   STATUS[640].EXT.AlarmPrsent := FALSE;
   STATUS[640].EXT.AlarmFailUnAck := FALSE;
   STATUS[640].Status := 0;
   STATUS[640].TimeStamp := 16#0000;
   STATUS[641].VALUE := 0.0;
   STATUS[641].TRIGVALUE := 0.0;
   STATUS[641].EXT.AlarmWarnUnAck := FALSE;
   STATUS[641].EXT.AckRequired := FALSE;
   STATUS[641].EXT.Maintanence := FALSE;
   STATUS[641].EXT.Operation := FALSE;
   STATUS[641].EXT.Forced := FALSE;
   STATUS[641].EXT.BIT29 := FALSE;
   STATUS[641].EXT.BIT30 := FALSE;
   STATUS[641].EXT.BIT31 := FALSE;
   STATUS[641].EXT.ModeBit1 := FALSE;
   STATUS[641].EXT.ModeBit2 := FALSE;
   STATUS[641].EXT.ModeBit3 := FALSE;
   STATUS[641].EXT.BIT19 := FALSE;
   STATUS[641].EXT.BIT20 := FALSE;
   STATUS[641].EXT.AlarmSuppressed := FALSE;
   STATUS[641].EXT.AlarmPrsent := FALSE;
   STATUS[641].EXT.AlarmFailUnAck := FALSE;
   STATUS[641].Status := 0;
   STATUS[641].TimeStamp := 16#0000;
   STATUS[642].VALUE := 0.0;
   STATUS[642].TRIGVALUE := 0.0;
   STATUS[642].EXT.AlarmWarnUnAck := FALSE;
   STATUS[642].EXT.AckRequired := FALSE;
   STATUS[642].EXT.Maintanence := FALSE;
   STATUS[642].EXT.Operation := FALSE;
   STATUS[642].EXT.Forced := FALSE;
   STATUS[642].EXT.BIT29 := FALSE;
   STATUS[642].EXT.BIT30 := FALSE;
   STATUS[642].EXT.BIT31 := FALSE;
   STATUS[642].EXT.ModeBit1 := FALSE;
   STATUS[642].EXT.ModeBit2 := FALSE;
   STATUS[642].EXT.ModeBit3 := FALSE;
   STATUS[642].EXT.BIT19 := FALSE;
   STATUS[642].EXT.BIT20 := FALSE;
   STATUS[642].EXT.AlarmSuppressed := FALSE;
   STATUS[642].EXT.AlarmPrsent := FALSE;
   STATUS[642].EXT.AlarmFailUnAck := FALSE;
   STATUS[642].Status := 0;
   STATUS[642].TimeStamp := 16#0000;
   STATUS[643].VALUE := 0.0;
   STATUS[643].TRIGVALUE := 0.0;
   STATUS[643].EXT.AlarmWarnUnAck := FALSE;
   STATUS[643].EXT.AckRequired := FALSE;
   STATUS[643].EXT.Maintanence := FALSE;
   STATUS[643].EXT.Operation := FALSE;
   STATUS[643].EXT.Forced := FALSE;
   STATUS[643].EXT.BIT29 := FALSE;
   STATUS[643].EXT.BIT30 := FALSE;
   STATUS[643].EXT.BIT31 := FALSE;
   STATUS[643].EXT.ModeBit1 := FALSE;
   STATUS[643].EXT.ModeBit2 := FALSE;
   STATUS[643].EXT.ModeBit3 := FALSE;
   STATUS[643].EXT.BIT19 := FALSE;
   STATUS[643].EXT.BIT20 := FALSE;
   STATUS[643].EXT.AlarmSuppressed := FALSE;
   STATUS[643].EXT.AlarmPrsent := FALSE;
   STATUS[643].EXT.AlarmFailUnAck := FALSE;
   STATUS[643].Status := 0;
   STATUS[643].TimeStamp := 16#0000;
   STATUS[644].VALUE := 0.0;
   STATUS[644].TRIGVALUE := 0.0;
   STATUS[644].EXT.AlarmWarnUnAck := FALSE;
   STATUS[644].EXT.AckRequired := FALSE;
   STATUS[644].EXT.Maintanence := FALSE;
   STATUS[644].EXT.Operation := FALSE;
   STATUS[644].EXT.Forced := FALSE;
   STATUS[644].EXT.BIT29 := FALSE;
   STATUS[644].EXT.BIT30 := FALSE;
   STATUS[644].EXT.BIT31 := FALSE;
   STATUS[644].EXT.ModeBit1 := FALSE;
   STATUS[644].EXT.ModeBit2 := FALSE;
   STATUS[644].EXT.ModeBit3 := FALSE;
   STATUS[644].EXT.BIT19 := FALSE;
   STATUS[644].EXT.BIT20 := FALSE;
   STATUS[644].EXT.AlarmSuppressed := FALSE;
   STATUS[644].EXT.AlarmPrsent := FALSE;
   STATUS[644].EXT.AlarmFailUnAck := FALSE;
   STATUS[644].Status := 0;
   STATUS[644].TimeStamp := 16#0000;
   STATUS[645].VALUE := 0.0;
   STATUS[645].TRIGVALUE := 0.0;
   STATUS[645].EXT.AlarmWarnUnAck := FALSE;
   STATUS[645].EXT.AckRequired := FALSE;
   STATUS[645].EXT.Maintanence := FALSE;
   STATUS[645].EXT.Operation := FALSE;
   STATUS[645].EXT.Forced := FALSE;
   STATUS[645].EXT.BIT29 := FALSE;
   STATUS[645].EXT.BIT30 := FALSE;
   STATUS[645].EXT.BIT31 := FALSE;
   STATUS[645].EXT.ModeBit1 := FALSE;
   STATUS[645].EXT.ModeBit2 := FALSE;
   STATUS[645].EXT.ModeBit3 := FALSE;
   STATUS[645].EXT.BIT19 := FALSE;
   STATUS[645].EXT.BIT20 := FALSE;
   STATUS[645].EXT.AlarmSuppressed := FALSE;
   STATUS[645].EXT.AlarmPrsent := FALSE;
   STATUS[645].EXT.AlarmFailUnAck := FALSE;
   STATUS[645].Status := 0;
   STATUS[645].TimeStamp := 16#0000;
   STATUS[646].VALUE := 0.0;
   STATUS[646].TRIGVALUE := 0.0;
   STATUS[646].EXT.AlarmWarnUnAck := FALSE;
   STATUS[646].EXT.AckRequired := FALSE;
   STATUS[646].EXT.Maintanence := FALSE;
   STATUS[646].EXT.Operation := FALSE;
   STATUS[646].EXT.Forced := FALSE;
   STATUS[646].EXT.BIT29 := FALSE;
   STATUS[646].EXT.BIT30 := FALSE;
   STATUS[646].EXT.BIT31 := FALSE;
   STATUS[646].EXT.ModeBit1 := FALSE;
   STATUS[646].EXT.ModeBit2 := FALSE;
   STATUS[646].EXT.ModeBit3 := FALSE;
   STATUS[646].EXT.BIT19 := FALSE;
   STATUS[646].EXT.BIT20 := FALSE;
   STATUS[646].EXT.AlarmSuppressed := FALSE;
   STATUS[646].EXT.AlarmPrsent := FALSE;
   STATUS[646].EXT.AlarmFailUnAck := FALSE;
   STATUS[646].Status := 0;
   STATUS[646].TimeStamp := 16#0000;
   STATUS[647].VALUE := 0.0;
   STATUS[647].TRIGVALUE := 0.0;
   STATUS[647].EXT.AlarmWarnUnAck := FALSE;
   STATUS[647].EXT.AckRequired := FALSE;
   STATUS[647].EXT.Maintanence := FALSE;
   STATUS[647].EXT.Operation := FALSE;
   STATUS[647].EXT.Forced := FALSE;
   STATUS[647].EXT.BIT29 := FALSE;
   STATUS[647].EXT.BIT30 := FALSE;
   STATUS[647].EXT.BIT31 := FALSE;
   STATUS[647].EXT.ModeBit1 := FALSE;
   STATUS[647].EXT.ModeBit2 := FALSE;
   STATUS[647].EXT.ModeBit3 := FALSE;
   STATUS[647].EXT.BIT19 := FALSE;
   STATUS[647].EXT.BIT20 := FALSE;
   STATUS[647].EXT.AlarmSuppressed := FALSE;
   STATUS[647].EXT.AlarmPrsent := FALSE;
   STATUS[647].EXT.AlarmFailUnAck := FALSE;
   STATUS[647].Status := 0;
   STATUS[647].TimeStamp := 16#0000;
   STATUS[648].VALUE := 0.0;
   STATUS[648].TRIGVALUE := 0.0;
   STATUS[648].EXT.AlarmWarnUnAck := FALSE;
   STATUS[648].EXT.AckRequired := FALSE;
   STATUS[648].EXT.Maintanence := FALSE;
   STATUS[648].EXT.Operation := FALSE;
   STATUS[648].EXT.Forced := FALSE;
   STATUS[648].EXT.BIT29 := FALSE;
   STATUS[648].EXT.BIT30 := FALSE;
   STATUS[648].EXT.BIT31 := FALSE;
   STATUS[648].EXT.ModeBit1 := FALSE;
   STATUS[648].EXT.ModeBit2 := FALSE;
   STATUS[648].EXT.ModeBit3 := FALSE;
   STATUS[648].EXT.BIT19 := FALSE;
   STATUS[648].EXT.BIT20 := FALSE;
   STATUS[648].EXT.AlarmSuppressed := FALSE;
   STATUS[648].EXT.AlarmPrsent := FALSE;
   STATUS[648].EXT.AlarmFailUnAck := FALSE;
   STATUS[648].Status := 0;
   STATUS[648].TimeStamp := 16#0000;
   STATUS[649].VALUE := 0.0;
   STATUS[649].TRIGVALUE := 0.0;
   STATUS[649].EXT.AlarmWarnUnAck := FALSE;
   STATUS[649].EXT.AckRequired := FALSE;
   STATUS[649].EXT.Maintanence := FALSE;
   STATUS[649].EXT.Operation := FALSE;
   STATUS[649].EXT.Forced := FALSE;
   STATUS[649].EXT.BIT29 := FALSE;
   STATUS[649].EXT.BIT30 := FALSE;
   STATUS[649].EXT.BIT31 := FALSE;
   STATUS[649].EXT.ModeBit1 := FALSE;
   STATUS[649].EXT.ModeBit2 := FALSE;
   STATUS[649].EXT.ModeBit3 := FALSE;
   STATUS[649].EXT.BIT19 := FALSE;
   STATUS[649].EXT.BIT20 := FALSE;
   STATUS[649].EXT.AlarmSuppressed := FALSE;
   STATUS[649].EXT.AlarmPrsent := FALSE;
   STATUS[649].EXT.AlarmFailUnAck := FALSE;
   STATUS[649].Status := 0;
   STATUS[649].TimeStamp := 16#0000;
   STATUS[650].VALUE := 0.0;
   STATUS[650].TRIGVALUE := 0.0;
   STATUS[650].EXT.AlarmWarnUnAck := FALSE;
   STATUS[650].EXT.AckRequired := FALSE;
   STATUS[650].EXT.Maintanence := FALSE;
   STATUS[650].EXT.Operation := FALSE;
   STATUS[650].EXT.Forced := FALSE;
   STATUS[650].EXT.BIT29 := FALSE;
   STATUS[650].EXT.BIT30 := FALSE;
   STATUS[650].EXT.BIT31 := FALSE;
   STATUS[650].EXT.ModeBit1 := FALSE;
   STATUS[650].EXT.ModeBit2 := FALSE;
   STATUS[650].EXT.ModeBit3 := FALSE;
   STATUS[650].EXT.BIT19 := FALSE;
   STATUS[650].EXT.BIT20 := FALSE;
   STATUS[650].EXT.AlarmSuppressed := FALSE;
   STATUS[650].EXT.AlarmPrsent := FALSE;
   STATUS[650].EXT.AlarmFailUnAck := FALSE;
   STATUS[650].Status := 0;
   STATUS[650].TimeStamp := 16#0000;
   STATUS[651].VALUE := 0.0;
   STATUS[651].TRIGVALUE := 0.0;
   STATUS[651].EXT.AlarmWarnUnAck := FALSE;
   STATUS[651].EXT.AckRequired := FALSE;
   STATUS[651].EXT.Maintanence := FALSE;
   STATUS[651].EXT.Operation := FALSE;
   STATUS[651].EXT.Forced := FALSE;
   STATUS[651].EXT.BIT29 := FALSE;
   STATUS[651].EXT.BIT30 := FALSE;
   STATUS[651].EXT.BIT31 := FALSE;
   STATUS[651].EXT.ModeBit1 := FALSE;
   STATUS[651].EXT.ModeBit2 := FALSE;
   STATUS[651].EXT.ModeBit3 := FALSE;
   STATUS[651].EXT.BIT19 := FALSE;
   STATUS[651].EXT.BIT20 := FALSE;
   STATUS[651].EXT.AlarmSuppressed := FALSE;
   STATUS[651].EXT.AlarmPrsent := FALSE;
   STATUS[651].EXT.AlarmFailUnAck := FALSE;
   STATUS[651].Status := 0;
   STATUS[651].TimeStamp := 16#0000;
   STATUS[652].VALUE := 0.0;
   STATUS[652].TRIGVALUE := 0.0;
   STATUS[652].EXT.AlarmWarnUnAck := FALSE;
   STATUS[652].EXT.AckRequired := FALSE;
   STATUS[652].EXT.Maintanence := FALSE;
   STATUS[652].EXT.Operation := FALSE;
   STATUS[652].EXT.Forced := FALSE;
   STATUS[652].EXT.BIT29 := FALSE;
   STATUS[652].EXT.BIT30 := FALSE;
   STATUS[652].EXT.BIT31 := FALSE;
   STATUS[652].EXT.ModeBit1 := FALSE;
   STATUS[652].EXT.ModeBit2 := FALSE;
   STATUS[652].EXT.ModeBit3 := FALSE;
   STATUS[652].EXT.BIT19 := FALSE;
   STATUS[652].EXT.BIT20 := FALSE;
   STATUS[652].EXT.AlarmSuppressed := FALSE;
   STATUS[652].EXT.AlarmPrsent := FALSE;
   STATUS[652].EXT.AlarmFailUnAck := FALSE;
   STATUS[652].Status := 0;
   STATUS[652].TimeStamp := 16#0000;
   STATUS[653].VALUE := 0.0;
   STATUS[653].TRIGVALUE := 0.0;
   STATUS[653].EXT.AlarmWarnUnAck := FALSE;
   STATUS[653].EXT.AckRequired := FALSE;
   STATUS[653].EXT.Maintanence := FALSE;
   STATUS[653].EXT.Operation := FALSE;
   STATUS[653].EXT.Forced := FALSE;
   STATUS[653].EXT.BIT29 := FALSE;
   STATUS[653].EXT.BIT30 := FALSE;
   STATUS[653].EXT.BIT31 := FALSE;
   STATUS[653].EXT.ModeBit1 := FALSE;
   STATUS[653].EXT.ModeBit2 := FALSE;
   STATUS[653].EXT.ModeBit3 := FALSE;
   STATUS[653].EXT.BIT19 := FALSE;
   STATUS[653].EXT.BIT20 := FALSE;
   STATUS[653].EXT.AlarmSuppressed := FALSE;
   STATUS[653].EXT.AlarmPrsent := FALSE;
   STATUS[653].EXT.AlarmFailUnAck := FALSE;
   STATUS[653].Status := 0;
   STATUS[653].TimeStamp := 16#0000;
   STATUS[654].VALUE := 0.0;
   STATUS[654].TRIGVALUE := 0.0;
   STATUS[654].EXT.AlarmWarnUnAck := FALSE;
   STATUS[654].EXT.AckRequired := FALSE;
   STATUS[654].EXT.Maintanence := FALSE;
   STATUS[654].EXT.Operation := FALSE;
   STATUS[654].EXT.Forced := FALSE;
   STATUS[654].EXT.BIT29 := FALSE;
   STATUS[654].EXT.BIT30 := FALSE;
   STATUS[654].EXT.BIT31 := FALSE;
   STATUS[654].EXT.ModeBit1 := FALSE;
   STATUS[654].EXT.ModeBit2 := FALSE;
   STATUS[654].EXT.ModeBit3 := FALSE;
   STATUS[654].EXT.BIT19 := FALSE;
   STATUS[654].EXT.BIT20 := FALSE;
   STATUS[654].EXT.AlarmSuppressed := FALSE;
   STATUS[654].EXT.AlarmPrsent := FALSE;
   STATUS[654].EXT.AlarmFailUnAck := FALSE;
   STATUS[654].Status := 0;
   STATUS[654].TimeStamp := 16#0000;
   STATUS[655].VALUE := 0.0;
   STATUS[655].TRIGVALUE := 0.0;
   STATUS[655].EXT.AlarmWarnUnAck := FALSE;
   STATUS[655].EXT.AckRequired := FALSE;
   STATUS[655].EXT.Maintanence := FALSE;
   STATUS[655].EXT.Operation := FALSE;
   STATUS[655].EXT.Forced := FALSE;
   STATUS[655].EXT.BIT29 := FALSE;
   STATUS[655].EXT.BIT30 := FALSE;
   STATUS[655].EXT.BIT31 := FALSE;
   STATUS[655].EXT.ModeBit1 := FALSE;
   STATUS[655].EXT.ModeBit2 := FALSE;
   STATUS[655].EXT.ModeBit3 := FALSE;
   STATUS[655].EXT.BIT19 := FALSE;
   STATUS[655].EXT.BIT20 := FALSE;
   STATUS[655].EXT.AlarmSuppressed := FALSE;
   STATUS[655].EXT.AlarmPrsent := FALSE;
   STATUS[655].EXT.AlarmFailUnAck := FALSE;
   STATUS[655].Status := 0;
   STATUS[655].TimeStamp := 16#0000;
   STATUS[656].VALUE := 0.0;
   STATUS[656].TRIGVALUE := 0.0;
   STATUS[656].EXT.AlarmWarnUnAck := FALSE;
   STATUS[656].EXT.AckRequired := FALSE;
   STATUS[656].EXT.Maintanence := FALSE;
   STATUS[656].EXT.Operation := FALSE;
   STATUS[656].EXT.Forced := FALSE;
   STATUS[656].EXT.BIT29 := FALSE;
   STATUS[656].EXT.BIT30 := FALSE;
   STATUS[656].EXT.BIT31 := FALSE;
   STATUS[656].EXT.ModeBit1 := FALSE;
   STATUS[656].EXT.ModeBit2 := FALSE;
   STATUS[656].EXT.ModeBit3 := FALSE;
   STATUS[656].EXT.BIT19 := FALSE;
   STATUS[656].EXT.BIT20 := FALSE;
   STATUS[656].EXT.AlarmSuppressed := FALSE;
   STATUS[656].EXT.AlarmPrsent := FALSE;
   STATUS[656].EXT.AlarmFailUnAck := FALSE;
   STATUS[656].Status := 0;
   STATUS[656].TimeStamp := 16#0000;
   STATUS[657].VALUE := 0.0;
   STATUS[657].TRIGVALUE := 0.0;
   STATUS[657].EXT.AlarmWarnUnAck := FALSE;
   STATUS[657].EXT.AckRequired := FALSE;
   STATUS[657].EXT.Maintanence := FALSE;
   STATUS[657].EXT.Operation := FALSE;
   STATUS[657].EXT.Forced := FALSE;
   STATUS[657].EXT.BIT29 := FALSE;
   STATUS[657].EXT.BIT30 := FALSE;
   STATUS[657].EXT.BIT31 := FALSE;
   STATUS[657].EXT.ModeBit1 := FALSE;
   STATUS[657].EXT.ModeBit2 := FALSE;
   STATUS[657].EXT.ModeBit3 := FALSE;
   STATUS[657].EXT.BIT19 := FALSE;
   STATUS[657].EXT.BIT20 := FALSE;
   STATUS[657].EXT.AlarmSuppressed := FALSE;
   STATUS[657].EXT.AlarmPrsent := FALSE;
   STATUS[657].EXT.AlarmFailUnAck := FALSE;
   STATUS[657].Status := 0;
   STATUS[657].TimeStamp := 16#0000;
   STATUS[658].VALUE := 0.0;
   STATUS[658].TRIGVALUE := 0.0;
   STATUS[658].EXT.AlarmWarnUnAck := FALSE;
   STATUS[658].EXT.AckRequired := FALSE;
   STATUS[658].EXT.Maintanence := FALSE;
   STATUS[658].EXT.Operation := FALSE;
   STATUS[658].EXT.Forced := FALSE;
   STATUS[658].EXT.BIT29 := FALSE;
   STATUS[658].EXT.BIT30 := FALSE;
   STATUS[658].EXT.BIT31 := FALSE;
   STATUS[658].EXT.ModeBit1 := FALSE;
   STATUS[658].EXT.ModeBit2 := FALSE;
   STATUS[658].EXT.ModeBit3 := FALSE;
   STATUS[658].EXT.BIT19 := FALSE;
   STATUS[658].EXT.BIT20 := FALSE;
   STATUS[658].EXT.AlarmSuppressed := FALSE;
   STATUS[658].EXT.AlarmPrsent := FALSE;
   STATUS[658].EXT.AlarmFailUnAck := FALSE;
   STATUS[658].Status := 0;
   STATUS[658].TimeStamp := 16#0000;
   STATUS[659].VALUE := 0.0;
   STATUS[659].TRIGVALUE := 0.0;
   STATUS[659].EXT.AlarmWarnUnAck := FALSE;
   STATUS[659].EXT.AckRequired := FALSE;
   STATUS[659].EXT.Maintanence := FALSE;
   STATUS[659].EXT.Operation := FALSE;
   STATUS[659].EXT.Forced := FALSE;
   STATUS[659].EXT.BIT29 := FALSE;
   STATUS[659].EXT.BIT30 := FALSE;
   STATUS[659].EXT.BIT31 := FALSE;
   STATUS[659].EXT.ModeBit1 := FALSE;
   STATUS[659].EXT.ModeBit2 := FALSE;
   STATUS[659].EXT.ModeBit3 := FALSE;
   STATUS[659].EXT.BIT19 := FALSE;
   STATUS[659].EXT.BIT20 := FALSE;
   STATUS[659].EXT.AlarmSuppressed := FALSE;
   STATUS[659].EXT.AlarmPrsent := FALSE;
   STATUS[659].EXT.AlarmFailUnAck := FALSE;
   STATUS[659].Status := 0;
   STATUS[659].TimeStamp := 16#0000;
   STATUS[660].VALUE := 0.0;
   STATUS[660].TRIGVALUE := 0.0;
   STATUS[660].EXT.AlarmWarnUnAck := FALSE;
   STATUS[660].EXT.AckRequired := FALSE;
   STATUS[660].EXT.Maintanence := FALSE;
   STATUS[660].EXT.Operation := FALSE;
   STATUS[660].EXT.Forced := FALSE;
   STATUS[660].EXT.BIT29 := FALSE;
   STATUS[660].EXT.BIT30 := FALSE;
   STATUS[660].EXT.BIT31 := FALSE;
   STATUS[660].EXT.ModeBit1 := FALSE;
   STATUS[660].EXT.ModeBit2 := FALSE;
   STATUS[660].EXT.ModeBit3 := FALSE;
   STATUS[660].EXT.BIT19 := FALSE;
   STATUS[660].EXT.BIT20 := FALSE;
   STATUS[660].EXT.AlarmSuppressed := FALSE;
   STATUS[660].EXT.AlarmPrsent := FALSE;
   STATUS[660].EXT.AlarmFailUnAck := FALSE;
   STATUS[660].Status := 0;
   STATUS[660].TimeStamp := 16#0000;
   STATUS[661].VALUE := 0.0;
   STATUS[661].TRIGVALUE := 0.0;
   STATUS[661].EXT.AlarmWarnUnAck := FALSE;
   STATUS[661].EXT.AckRequired := FALSE;
   STATUS[661].EXT.Maintanence := FALSE;
   STATUS[661].EXT.Operation := FALSE;
   STATUS[661].EXT.Forced := FALSE;
   STATUS[661].EXT.BIT29 := FALSE;
   STATUS[661].EXT.BIT30 := FALSE;
   STATUS[661].EXT.BIT31 := FALSE;
   STATUS[661].EXT.ModeBit1 := FALSE;
   STATUS[661].EXT.ModeBit2 := FALSE;
   STATUS[661].EXT.ModeBit3 := FALSE;
   STATUS[661].EXT.BIT19 := FALSE;
   STATUS[661].EXT.BIT20 := FALSE;
   STATUS[661].EXT.AlarmSuppressed := FALSE;
   STATUS[661].EXT.AlarmPrsent := FALSE;
   STATUS[661].EXT.AlarmFailUnAck := FALSE;
   STATUS[661].Status := 0;
   STATUS[661].TimeStamp := 16#0000;
   STATUS[662].VALUE := 0.0;
   STATUS[662].TRIGVALUE := 0.0;
   STATUS[662].EXT.AlarmWarnUnAck := FALSE;
   STATUS[662].EXT.AckRequired := FALSE;
   STATUS[662].EXT.Maintanence := FALSE;
   STATUS[662].EXT.Operation := FALSE;
   STATUS[662].EXT.Forced := FALSE;
   STATUS[662].EXT.BIT29 := FALSE;
   STATUS[662].EXT.BIT30 := FALSE;
   STATUS[662].EXT.BIT31 := FALSE;
   STATUS[662].EXT.ModeBit1 := FALSE;
   STATUS[662].EXT.ModeBit2 := FALSE;
   STATUS[662].EXT.ModeBit3 := FALSE;
   STATUS[662].EXT.BIT19 := FALSE;
   STATUS[662].EXT.BIT20 := FALSE;
   STATUS[662].EXT.AlarmSuppressed := FALSE;
   STATUS[662].EXT.AlarmPrsent := FALSE;
   STATUS[662].EXT.AlarmFailUnAck := FALSE;
   STATUS[662].Status := 0;
   STATUS[662].TimeStamp := 16#0000;
   STATUS[663].VALUE := 0.0;
   STATUS[663].TRIGVALUE := 0.0;
   STATUS[663].EXT.AlarmWarnUnAck := FALSE;
   STATUS[663].EXT.AckRequired := FALSE;
   STATUS[663].EXT.Maintanence := FALSE;
   STATUS[663].EXT.Operation := FALSE;
   STATUS[663].EXT.Forced := FALSE;
   STATUS[663].EXT.BIT29 := FALSE;
   STATUS[663].EXT.BIT30 := FALSE;
   STATUS[663].EXT.BIT31 := FALSE;
   STATUS[663].EXT.ModeBit1 := FALSE;
   STATUS[663].EXT.ModeBit2 := FALSE;
   STATUS[663].EXT.ModeBit3 := FALSE;
   STATUS[663].EXT.BIT19 := FALSE;
   STATUS[663].EXT.BIT20 := FALSE;
   STATUS[663].EXT.AlarmSuppressed := FALSE;
   STATUS[663].EXT.AlarmPrsent := FALSE;
   STATUS[663].EXT.AlarmFailUnAck := FALSE;
   STATUS[663].Status := 0;
   STATUS[663].TimeStamp := 16#0000;
   STATUS[664].VALUE := 0.0;
   STATUS[664].TRIGVALUE := 0.0;
   STATUS[664].EXT.AlarmWarnUnAck := FALSE;
   STATUS[664].EXT.AckRequired := FALSE;
   STATUS[664].EXT.Maintanence := FALSE;
   STATUS[664].EXT.Operation := FALSE;
   STATUS[664].EXT.Forced := FALSE;
   STATUS[664].EXT.BIT29 := FALSE;
   STATUS[664].EXT.BIT30 := FALSE;
   STATUS[664].EXT.BIT31 := FALSE;
   STATUS[664].EXT.ModeBit1 := FALSE;
   STATUS[664].EXT.ModeBit2 := FALSE;
   STATUS[664].EXT.ModeBit3 := FALSE;
   STATUS[664].EXT.BIT19 := FALSE;
   STATUS[664].EXT.BIT20 := FALSE;
   STATUS[664].EXT.AlarmSuppressed := FALSE;
   STATUS[664].EXT.AlarmPrsent := FALSE;
   STATUS[664].EXT.AlarmFailUnAck := FALSE;
   STATUS[664].Status := 0;
   STATUS[664].TimeStamp := 16#0000;
   STATUS[665].VALUE := 0.0;
   STATUS[665].TRIGVALUE := 0.0;
   STATUS[665].EXT.AlarmWarnUnAck := FALSE;
   STATUS[665].EXT.AckRequired := FALSE;
   STATUS[665].EXT.Maintanence := FALSE;
   STATUS[665].EXT.Operation := FALSE;
   STATUS[665].EXT.Forced := FALSE;
   STATUS[665].EXT.BIT29 := FALSE;
   STATUS[665].EXT.BIT30 := FALSE;
   STATUS[665].EXT.BIT31 := FALSE;
   STATUS[665].EXT.ModeBit1 := FALSE;
   STATUS[665].EXT.ModeBit2 := FALSE;
   STATUS[665].EXT.ModeBit3 := FALSE;
   STATUS[665].EXT.BIT19 := FALSE;
   STATUS[665].EXT.BIT20 := FALSE;
   STATUS[665].EXT.AlarmSuppressed := FALSE;
   STATUS[665].EXT.AlarmPrsent := FALSE;
   STATUS[665].EXT.AlarmFailUnAck := FALSE;
   STATUS[665].Status := 0;
   STATUS[665].TimeStamp := 16#0000;
   STATUS[666].VALUE := 0.0;
   STATUS[666].TRIGVALUE := 0.0;
   STATUS[666].EXT.AlarmWarnUnAck := FALSE;
   STATUS[666].EXT.AckRequired := FALSE;
   STATUS[666].EXT.Maintanence := FALSE;
   STATUS[666].EXT.Operation := FALSE;
   STATUS[666].EXT.Forced := FALSE;
   STATUS[666].EXT.BIT29 := FALSE;
   STATUS[666].EXT.BIT30 := FALSE;
   STATUS[666].EXT.BIT31 := FALSE;
   STATUS[666].EXT.ModeBit1 := FALSE;
   STATUS[666].EXT.ModeBit2 := FALSE;
   STATUS[666].EXT.ModeBit3 := FALSE;
   STATUS[666].EXT.BIT19 := FALSE;
   STATUS[666].EXT.BIT20 := FALSE;
   STATUS[666].EXT.AlarmSuppressed := FALSE;
   STATUS[666].EXT.AlarmPrsent := FALSE;
   STATUS[666].EXT.AlarmFailUnAck := FALSE;
   STATUS[666].Status := 0;
   STATUS[666].TimeStamp := 16#0000;
   STATUS[667].VALUE := 0.0;
   STATUS[667].TRIGVALUE := 0.0;
   STATUS[667].EXT.AlarmWarnUnAck := FALSE;
   STATUS[667].EXT.AckRequired := FALSE;
   STATUS[667].EXT.Maintanence := FALSE;
   STATUS[667].EXT.Operation := FALSE;
   STATUS[667].EXT.Forced := FALSE;
   STATUS[667].EXT.BIT29 := FALSE;
   STATUS[667].EXT.BIT30 := FALSE;
   STATUS[667].EXT.BIT31 := FALSE;
   STATUS[667].EXT.ModeBit1 := FALSE;
   STATUS[667].EXT.ModeBit2 := FALSE;
   STATUS[667].EXT.ModeBit3 := FALSE;
   STATUS[667].EXT.BIT19 := FALSE;
   STATUS[667].EXT.BIT20 := FALSE;
   STATUS[667].EXT.AlarmSuppressed := FALSE;
   STATUS[667].EXT.AlarmPrsent := FALSE;
   STATUS[667].EXT.AlarmFailUnAck := FALSE;
   STATUS[667].Status := 0;
   STATUS[667].TimeStamp := 16#0000;
   STATUS[668].VALUE := 0.0;
   STATUS[668].TRIGVALUE := 0.0;
   STATUS[668].EXT.AlarmWarnUnAck := FALSE;
   STATUS[668].EXT.AckRequired := FALSE;
   STATUS[668].EXT.Maintanence := FALSE;
   STATUS[668].EXT.Operation := FALSE;
   STATUS[668].EXT.Forced := FALSE;
   STATUS[668].EXT.BIT29 := FALSE;
   STATUS[668].EXT.BIT30 := FALSE;
   STATUS[668].EXT.BIT31 := FALSE;
   STATUS[668].EXT.ModeBit1 := FALSE;
   STATUS[668].EXT.ModeBit2 := FALSE;
   STATUS[668].EXT.ModeBit3 := FALSE;
   STATUS[668].EXT.BIT19 := FALSE;
   STATUS[668].EXT.BIT20 := FALSE;
   STATUS[668].EXT.AlarmSuppressed := FALSE;
   STATUS[668].EXT.AlarmPrsent := FALSE;
   STATUS[668].EXT.AlarmFailUnAck := FALSE;
   STATUS[668].Status := 0;
   STATUS[668].TimeStamp := 16#0000;
   STATUS[669].VALUE := 0.0;
   STATUS[669].TRIGVALUE := 0.0;
   STATUS[669].EXT.AlarmWarnUnAck := FALSE;
   STATUS[669].EXT.AckRequired := FALSE;
   STATUS[669].EXT.Maintanence := FALSE;
   STATUS[669].EXT.Operation := FALSE;
   STATUS[669].EXT.Forced := FALSE;
   STATUS[669].EXT.BIT29 := FALSE;
   STATUS[669].EXT.BIT30 := FALSE;
   STATUS[669].EXT.BIT31 := FALSE;
   STATUS[669].EXT.ModeBit1 := FALSE;
   STATUS[669].EXT.ModeBit2 := FALSE;
   STATUS[669].EXT.ModeBit3 := FALSE;
   STATUS[669].EXT.BIT19 := FALSE;
   STATUS[669].EXT.BIT20 := FALSE;
   STATUS[669].EXT.AlarmSuppressed := FALSE;
   STATUS[669].EXT.AlarmPrsent := FALSE;
   STATUS[669].EXT.AlarmFailUnAck := FALSE;
   STATUS[669].Status := 0;
   STATUS[669].TimeStamp := 16#0000;
   STATUS[670].VALUE := 0.0;
   STATUS[670].TRIGVALUE := 0.0;
   STATUS[670].EXT.AlarmWarnUnAck := FALSE;
   STATUS[670].EXT.AckRequired := FALSE;
   STATUS[670].EXT.Maintanence := FALSE;
   STATUS[670].EXT.Operation := FALSE;
   STATUS[670].EXT.Forced := FALSE;
   STATUS[670].EXT.BIT29 := FALSE;
   STATUS[670].EXT.BIT30 := FALSE;
   STATUS[670].EXT.BIT31 := FALSE;
   STATUS[670].EXT.ModeBit1 := FALSE;
   STATUS[670].EXT.ModeBit2 := FALSE;
   STATUS[670].EXT.ModeBit3 := FALSE;
   STATUS[670].EXT.BIT19 := FALSE;
   STATUS[670].EXT.BIT20 := FALSE;
   STATUS[670].EXT.AlarmSuppressed := FALSE;
   STATUS[670].EXT.AlarmPrsent := FALSE;
   STATUS[670].EXT.AlarmFailUnAck := FALSE;
   STATUS[670].Status := 0;
   STATUS[670].TimeStamp := 16#0000;
   STATUS[671].VALUE := 0.0;
   STATUS[671].TRIGVALUE := 0.0;
   STATUS[671].EXT.AlarmWarnUnAck := FALSE;
   STATUS[671].EXT.AckRequired := FALSE;
   STATUS[671].EXT.Maintanence := FALSE;
   STATUS[671].EXT.Operation := FALSE;
   STATUS[671].EXT.Forced := FALSE;
   STATUS[671].EXT.BIT29 := FALSE;
   STATUS[671].EXT.BIT30 := FALSE;
   STATUS[671].EXT.BIT31 := FALSE;
   STATUS[671].EXT.ModeBit1 := FALSE;
   STATUS[671].EXT.ModeBit2 := FALSE;
   STATUS[671].EXT.ModeBit3 := FALSE;
   STATUS[671].EXT.BIT19 := FALSE;
   STATUS[671].EXT.BIT20 := FALSE;
   STATUS[671].EXT.AlarmSuppressed := FALSE;
   STATUS[671].EXT.AlarmPrsent := FALSE;
   STATUS[671].EXT.AlarmFailUnAck := FALSE;
   STATUS[671].Status := 0;
   STATUS[671].TimeStamp := 16#0000;
   STATUS[672].VALUE := 0.0;
   STATUS[672].TRIGVALUE := 0.0;
   STATUS[672].EXT.AlarmWarnUnAck := FALSE;
   STATUS[672].EXT.AckRequired := FALSE;
   STATUS[672].EXT.Maintanence := FALSE;
   STATUS[672].EXT.Operation := FALSE;
   STATUS[672].EXT.Forced := FALSE;
   STATUS[672].EXT.BIT29 := FALSE;
   STATUS[672].EXT.BIT30 := FALSE;
   STATUS[672].EXT.BIT31 := FALSE;
   STATUS[672].EXT.ModeBit1 := FALSE;
   STATUS[672].EXT.ModeBit2 := FALSE;
   STATUS[672].EXT.ModeBit3 := FALSE;
   STATUS[672].EXT.BIT19 := FALSE;
   STATUS[672].EXT.BIT20 := FALSE;
   STATUS[672].EXT.AlarmSuppressed := FALSE;
   STATUS[672].EXT.AlarmPrsent := FALSE;
   STATUS[672].EXT.AlarmFailUnAck := FALSE;
   STATUS[672].Status := 0;
   STATUS[672].TimeStamp := 16#0000;
   STATUS[673].VALUE := 0.0;
   STATUS[673].TRIGVALUE := 0.0;
   STATUS[673].EXT.AlarmWarnUnAck := FALSE;
   STATUS[673].EXT.AckRequired := FALSE;
   STATUS[673].EXT.Maintanence := FALSE;
   STATUS[673].EXT.Operation := FALSE;
   STATUS[673].EXT.Forced := FALSE;
   STATUS[673].EXT.BIT29 := FALSE;
   STATUS[673].EXT.BIT30 := FALSE;
   STATUS[673].EXT.BIT31 := FALSE;
   STATUS[673].EXT.ModeBit1 := FALSE;
   STATUS[673].EXT.ModeBit2 := FALSE;
   STATUS[673].EXT.ModeBit3 := FALSE;
   STATUS[673].EXT.BIT19 := FALSE;
   STATUS[673].EXT.BIT20 := FALSE;
   STATUS[673].EXT.AlarmSuppressed := FALSE;
   STATUS[673].EXT.AlarmPrsent := FALSE;
   STATUS[673].EXT.AlarmFailUnAck := FALSE;
   STATUS[673].Status := 0;
   STATUS[673].TimeStamp := 16#0000;
   STATUS[674].VALUE := 0.0;
   STATUS[674].TRIGVALUE := 0.0;
   STATUS[674].EXT.AlarmWarnUnAck := FALSE;
   STATUS[674].EXT.AckRequired := FALSE;
   STATUS[674].EXT.Maintanence := FALSE;
   STATUS[674].EXT.Operation := FALSE;
   STATUS[674].EXT.Forced := FALSE;
   STATUS[674].EXT.BIT29 := FALSE;
   STATUS[674].EXT.BIT30 := FALSE;
   STATUS[674].EXT.BIT31 := FALSE;
   STATUS[674].EXT.ModeBit1 := FALSE;
   STATUS[674].EXT.ModeBit2 := FALSE;
   STATUS[674].EXT.ModeBit3 := FALSE;
   STATUS[674].EXT.BIT19 := FALSE;
   STATUS[674].EXT.BIT20 := FALSE;
   STATUS[674].EXT.AlarmSuppressed := FALSE;
   STATUS[674].EXT.AlarmPrsent := FALSE;
   STATUS[674].EXT.AlarmFailUnAck := FALSE;
   STATUS[674].Status := 0;
   STATUS[674].TimeStamp := 16#0000;
   STATUS[675].VALUE := 0.0;
   STATUS[675].TRIGVALUE := 0.0;
   STATUS[675].EXT.AlarmWarnUnAck := FALSE;
   STATUS[675].EXT.AckRequired := FALSE;
   STATUS[675].EXT.Maintanence := FALSE;
   STATUS[675].EXT.Operation := FALSE;
   STATUS[675].EXT.Forced := FALSE;
   STATUS[675].EXT.BIT29 := FALSE;
   STATUS[675].EXT.BIT30 := FALSE;
   STATUS[675].EXT.BIT31 := FALSE;
   STATUS[675].EXT.ModeBit1 := FALSE;
   STATUS[675].EXT.ModeBit2 := FALSE;
   STATUS[675].EXT.ModeBit3 := FALSE;
   STATUS[675].EXT.BIT19 := FALSE;
   STATUS[675].EXT.BIT20 := FALSE;
   STATUS[675].EXT.AlarmSuppressed := FALSE;
   STATUS[675].EXT.AlarmPrsent := FALSE;
   STATUS[675].EXT.AlarmFailUnAck := FALSE;
   STATUS[675].Status := 0;
   STATUS[675].TimeStamp := 16#0000;
   STATUS[676].VALUE := 0.0;
   STATUS[676].TRIGVALUE := 0.0;
   STATUS[676].EXT.AlarmWarnUnAck := FALSE;
   STATUS[676].EXT.AckRequired := FALSE;
   STATUS[676].EXT.Maintanence := FALSE;
   STATUS[676].EXT.Operation := FALSE;
   STATUS[676].EXT.Forced := FALSE;
   STATUS[676].EXT.BIT29 := FALSE;
   STATUS[676].EXT.BIT30 := FALSE;
   STATUS[676].EXT.BIT31 := FALSE;
   STATUS[676].EXT.ModeBit1 := FALSE;
   STATUS[676].EXT.ModeBit2 := FALSE;
   STATUS[676].EXT.ModeBit3 := FALSE;
   STATUS[676].EXT.BIT19 := FALSE;
   STATUS[676].EXT.BIT20 := FALSE;
   STATUS[676].EXT.AlarmSuppressed := FALSE;
   STATUS[676].EXT.AlarmPrsent := FALSE;
   STATUS[676].EXT.AlarmFailUnAck := FALSE;
   STATUS[676].Status := 0;
   STATUS[676].TimeStamp := 16#0000;
   STATUS[677].VALUE := 0.0;
   STATUS[677].TRIGVALUE := 0.0;
   STATUS[677].EXT.AlarmWarnUnAck := FALSE;
   STATUS[677].EXT.AckRequired := FALSE;
   STATUS[677].EXT.Maintanence := FALSE;
   STATUS[677].EXT.Operation := FALSE;
   STATUS[677].EXT.Forced := FALSE;
   STATUS[677].EXT.BIT29 := FALSE;
   STATUS[677].EXT.BIT30 := FALSE;
   STATUS[677].EXT.BIT31 := FALSE;
   STATUS[677].EXT.ModeBit1 := FALSE;
   STATUS[677].EXT.ModeBit2 := FALSE;
   STATUS[677].EXT.ModeBit3 := FALSE;
   STATUS[677].EXT.BIT19 := FALSE;
   STATUS[677].EXT.BIT20 := FALSE;
   STATUS[677].EXT.AlarmSuppressed := FALSE;
   STATUS[677].EXT.AlarmPrsent := FALSE;
   STATUS[677].EXT.AlarmFailUnAck := FALSE;
   STATUS[677].Status := 0;
   STATUS[677].TimeStamp := 16#0000;
   STATUS[678].VALUE := 0.0;
   STATUS[678].TRIGVALUE := 0.0;
   STATUS[678].EXT.AlarmWarnUnAck := FALSE;
   STATUS[678].EXT.AckRequired := FALSE;
   STATUS[678].EXT.Maintanence := FALSE;
   STATUS[678].EXT.Operation := FALSE;
   STATUS[678].EXT.Forced := FALSE;
   STATUS[678].EXT.BIT29 := FALSE;
   STATUS[678].EXT.BIT30 := FALSE;
   STATUS[678].EXT.BIT31 := FALSE;
   STATUS[678].EXT.ModeBit1 := FALSE;
   STATUS[678].EXT.ModeBit2 := FALSE;
   STATUS[678].EXT.ModeBit3 := FALSE;
   STATUS[678].EXT.BIT19 := FALSE;
   STATUS[678].EXT.BIT20 := FALSE;
   STATUS[678].EXT.AlarmSuppressed := FALSE;
   STATUS[678].EXT.AlarmPrsent := FALSE;
   STATUS[678].EXT.AlarmFailUnAck := FALSE;
   STATUS[678].Status := 0;
   STATUS[678].TimeStamp := 16#0000;
   STATUS[679].VALUE := 0.0;
   STATUS[679].TRIGVALUE := 0.0;
   STATUS[679].EXT.AlarmWarnUnAck := FALSE;
   STATUS[679].EXT.AckRequired := FALSE;
   STATUS[679].EXT.Maintanence := FALSE;
   STATUS[679].EXT.Operation := FALSE;
   STATUS[679].EXT.Forced := FALSE;
   STATUS[679].EXT.BIT29 := FALSE;
   STATUS[679].EXT.BIT30 := FALSE;
   STATUS[679].EXT.BIT31 := FALSE;
   STATUS[679].EXT.ModeBit1 := FALSE;
   STATUS[679].EXT.ModeBit2 := FALSE;
   STATUS[679].EXT.ModeBit3 := FALSE;
   STATUS[679].EXT.BIT19 := FALSE;
   STATUS[679].EXT.BIT20 := FALSE;
   STATUS[679].EXT.AlarmSuppressed := FALSE;
   STATUS[679].EXT.AlarmPrsent := FALSE;
   STATUS[679].EXT.AlarmFailUnAck := FALSE;
   STATUS[679].Status := 0;
   STATUS[679].TimeStamp := 16#0000;
   STATUS[680].VALUE := 0.0;
   STATUS[680].TRIGVALUE := 0.0;
   STATUS[680].EXT.AlarmWarnUnAck := FALSE;
   STATUS[680].EXT.AckRequired := FALSE;
   STATUS[680].EXT.Maintanence := FALSE;
   STATUS[680].EXT.Operation := FALSE;
   STATUS[680].EXT.Forced := FALSE;
   STATUS[680].EXT.BIT29 := FALSE;
   STATUS[680].EXT.BIT30 := FALSE;
   STATUS[680].EXT.BIT31 := FALSE;
   STATUS[680].EXT.ModeBit1 := FALSE;
   STATUS[680].EXT.ModeBit2 := FALSE;
   STATUS[680].EXT.ModeBit3 := FALSE;
   STATUS[680].EXT.BIT19 := FALSE;
   STATUS[680].EXT.BIT20 := FALSE;
   STATUS[680].EXT.AlarmSuppressed := FALSE;
   STATUS[680].EXT.AlarmPrsent := FALSE;
   STATUS[680].EXT.AlarmFailUnAck := FALSE;
   STATUS[680].Status := 0;
   STATUS[680].TimeStamp := 16#0000;
   STATUS[681].VALUE := 0.0;
   STATUS[681].TRIGVALUE := 0.0;
   STATUS[681].EXT.AlarmWarnUnAck := FALSE;
   STATUS[681].EXT.AckRequired := FALSE;
   STATUS[681].EXT.Maintanence := FALSE;
   STATUS[681].EXT.Operation := FALSE;
   STATUS[681].EXT.Forced := FALSE;
   STATUS[681].EXT.BIT29 := FALSE;
   STATUS[681].EXT.BIT30 := FALSE;
   STATUS[681].EXT.BIT31 := FALSE;
   STATUS[681].EXT.ModeBit1 := FALSE;
   STATUS[681].EXT.ModeBit2 := FALSE;
   STATUS[681].EXT.ModeBit3 := FALSE;
   STATUS[681].EXT.BIT19 := FALSE;
   STATUS[681].EXT.BIT20 := FALSE;
   STATUS[681].EXT.AlarmSuppressed := FALSE;
   STATUS[681].EXT.AlarmPrsent := FALSE;
   STATUS[681].EXT.AlarmFailUnAck := FALSE;
   STATUS[681].Status := 0;
   STATUS[681].TimeStamp := 16#0000;
   STATUS[682].VALUE := 0.0;
   STATUS[682].TRIGVALUE := 0.0;
   STATUS[682].EXT.AlarmWarnUnAck := FALSE;
   STATUS[682].EXT.AckRequired := FALSE;
   STATUS[682].EXT.Maintanence := FALSE;
   STATUS[682].EXT.Operation := FALSE;
   STATUS[682].EXT.Forced := FALSE;
   STATUS[682].EXT.BIT29 := FALSE;
   STATUS[682].EXT.BIT30 := FALSE;
   STATUS[682].EXT.BIT31 := FALSE;
   STATUS[682].EXT.ModeBit1 := FALSE;
   STATUS[682].EXT.ModeBit2 := FALSE;
   STATUS[682].EXT.ModeBit3 := FALSE;
   STATUS[682].EXT.BIT19 := FALSE;
   STATUS[682].EXT.BIT20 := FALSE;
   STATUS[682].EXT.AlarmSuppressed := FALSE;
   STATUS[682].EXT.AlarmPrsent := FALSE;
   STATUS[682].EXT.AlarmFailUnAck := FALSE;
   STATUS[682].Status := 0;
   STATUS[682].TimeStamp := 16#0000;
   STATUS[683].VALUE := 0.0;
   STATUS[683].TRIGVALUE := 0.0;
   STATUS[683].EXT.AlarmWarnUnAck := FALSE;
   STATUS[683].EXT.AckRequired := FALSE;
   STATUS[683].EXT.Maintanence := FALSE;
   STATUS[683].EXT.Operation := FALSE;
   STATUS[683].EXT.Forced := FALSE;
   STATUS[683].EXT.BIT29 := FALSE;
   STATUS[683].EXT.BIT30 := FALSE;
   STATUS[683].EXT.BIT31 := FALSE;
   STATUS[683].EXT.ModeBit1 := FALSE;
   STATUS[683].EXT.ModeBit2 := FALSE;
   STATUS[683].EXT.ModeBit3 := FALSE;
   STATUS[683].EXT.BIT19 := FALSE;
   STATUS[683].EXT.BIT20 := FALSE;
   STATUS[683].EXT.AlarmSuppressed := FALSE;
   STATUS[683].EXT.AlarmPrsent := FALSE;
   STATUS[683].EXT.AlarmFailUnAck := FALSE;
   STATUS[683].Status := 0;
   STATUS[683].TimeStamp := 16#0000;
   STATUS[684].VALUE := 0.0;
   STATUS[684].TRIGVALUE := 0.0;
   STATUS[684].EXT.AlarmWarnUnAck := FALSE;
   STATUS[684].EXT.AckRequired := FALSE;
   STATUS[684].EXT.Maintanence := FALSE;
   STATUS[684].EXT.Operation := FALSE;
   STATUS[684].EXT.Forced := FALSE;
   STATUS[684].EXT.BIT29 := FALSE;
   STATUS[684].EXT.BIT30 := FALSE;
   STATUS[684].EXT.BIT31 := FALSE;
   STATUS[684].EXT.ModeBit1 := FALSE;
   STATUS[684].EXT.ModeBit2 := FALSE;
   STATUS[684].EXT.ModeBit3 := FALSE;
   STATUS[684].EXT.BIT19 := FALSE;
   STATUS[684].EXT.BIT20 := FALSE;
   STATUS[684].EXT.AlarmSuppressed := FALSE;
   STATUS[684].EXT.AlarmPrsent := FALSE;
   STATUS[684].EXT.AlarmFailUnAck := FALSE;
   STATUS[684].Status := 0;
   STATUS[684].TimeStamp := 16#0000;
   STATUS[685].VALUE := 0.0;
   STATUS[685].TRIGVALUE := 0.0;
   STATUS[685].EXT.AlarmWarnUnAck := FALSE;
   STATUS[685].EXT.AckRequired := FALSE;
   STATUS[685].EXT.Maintanence := FALSE;
   STATUS[685].EXT.Operation := FALSE;
   STATUS[685].EXT.Forced := FALSE;
   STATUS[685].EXT.BIT29 := FALSE;
   STATUS[685].EXT.BIT30 := FALSE;
   STATUS[685].EXT.BIT31 := FALSE;
   STATUS[685].EXT.ModeBit1 := FALSE;
   STATUS[685].EXT.ModeBit2 := FALSE;
   STATUS[685].EXT.ModeBit3 := FALSE;
   STATUS[685].EXT.BIT19 := FALSE;
   STATUS[685].EXT.BIT20 := FALSE;
   STATUS[685].EXT.AlarmSuppressed := FALSE;
   STATUS[685].EXT.AlarmPrsent := FALSE;
   STATUS[685].EXT.AlarmFailUnAck := FALSE;
   STATUS[685].Status := 0;
   STATUS[685].TimeStamp := 16#0000;
   STATUS[686].VALUE := 0.0;
   STATUS[686].TRIGVALUE := 0.0;
   STATUS[686].EXT.AlarmWarnUnAck := FALSE;
   STATUS[686].EXT.AckRequired := FALSE;
   STATUS[686].EXT.Maintanence := FALSE;
   STATUS[686].EXT.Operation := FALSE;
   STATUS[686].EXT.Forced := FALSE;
   STATUS[686].EXT.BIT29 := FALSE;
   STATUS[686].EXT.BIT30 := FALSE;
   STATUS[686].EXT.BIT31 := FALSE;
   STATUS[686].EXT.ModeBit1 := FALSE;
   STATUS[686].EXT.ModeBit2 := FALSE;
   STATUS[686].EXT.ModeBit3 := FALSE;
   STATUS[686].EXT.BIT19 := FALSE;
   STATUS[686].EXT.BIT20 := FALSE;
   STATUS[686].EXT.AlarmSuppressed := FALSE;
   STATUS[686].EXT.AlarmPrsent := FALSE;
   STATUS[686].EXT.AlarmFailUnAck := FALSE;
   STATUS[686].Status := 0;
   STATUS[686].TimeStamp := 16#0000;
   STATUS[687].VALUE := 0.0;
   STATUS[687].TRIGVALUE := 0.0;
   STATUS[687].EXT.AlarmWarnUnAck := FALSE;
   STATUS[687].EXT.AckRequired := FALSE;
   STATUS[687].EXT.Maintanence := FALSE;
   STATUS[687].EXT.Operation := FALSE;
   STATUS[687].EXT.Forced := FALSE;
   STATUS[687].EXT.BIT29 := FALSE;
   STATUS[687].EXT.BIT30 := FALSE;
   STATUS[687].EXT.BIT31 := FALSE;
   STATUS[687].EXT.ModeBit1 := FALSE;
   STATUS[687].EXT.ModeBit2 := FALSE;
   STATUS[687].EXT.ModeBit3 := FALSE;
   STATUS[687].EXT.BIT19 := FALSE;
   STATUS[687].EXT.BIT20 := FALSE;
   STATUS[687].EXT.AlarmSuppressed := FALSE;
   STATUS[687].EXT.AlarmPrsent := FALSE;
   STATUS[687].EXT.AlarmFailUnAck := FALSE;
   STATUS[687].Status := 0;
   STATUS[687].TimeStamp := 16#0000;
   STATUS[688].VALUE := 0.0;
   STATUS[688].TRIGVALUE := 0.0;
   STATUS[688].EXT.AlarmWarnUnAck := FALSE;
   STATUS[688].EXT.AckRequired := FALSE;
   STATUS[688].EXT.Maintanence := FALSE;
   STATUS[688].EXT.Operation := FALSE;
   STATUS[688].EXT.Forced := FALSE;
   STATUS[688].EXT.BIT29 := FALSE;
   STATUS[688].EXT.BIT30 := FALSE;
   STATUS[688].EXT.BIT31 := FALSE;
   STATUS[688].EXT.ModeBit1 := FALSE;
   STATUS[688].EXT.ModeBit2 := FALSE;
   STATUS[688].EXT.ModeBit3 := FALSE;
   STATUS[688].EXT.BIT19 := FALSE;
   STATUS[688].EXT.BIT20 := FALSE;
   STATUS[688].EXT.AlarmSuppressed := FALSE;
   STATUS[688].EXT.AlarmPrsent := FALSE;
   STATUS[688].EXT.AlarmFailUnAck := FALSE;
   STATUS[688].Status := 0;
   STATUS[688].TimeStamp := 16#0000;
   STATUS[689].VALUE := 0.0;
   STATUS[689].TRIGVALUE := 0.0;
   STATUS[689].EXT.AlarmWarnUnAck := FALSE;
   STATUS[689].EXT.AckRequired := FALSE;
   STATUS[689].EXT.Maintanence := FALSE;
   STATUS[689].EXT.Operation := FALSE;
   STATUS[689].EXT.Forced := FALSE;
   STATUS[689].EXT.BIT29 := FALSE;
   STATUS[689].EXT.BIT30 := FALSE;
   STATUS[689].EXT.BIT31 := FALSE;
   STATUS[689].EXT.ModeBit1 := FALSE;
   STATUS[689].EXT.ModeBit2 := FALSE;
   STATUS[689].EXT.ModeBit3 := FALSE;
   STATUS[689].EXT.BIT19 := FALSE;
   STATUS[689].EXT.BIT20 := FALSE;
   STATUS[689].EXT.AlarmSuppressed := FALSE;
   STATUS[689].EXT.AlarmPrsent := FALSE;
   STATUS[689].EXT.AlarmFailUnAck := FALSE;
   STATUS[689].Status := 0;
   STATUS[689].TimeStamp := 16#0000;
   STATUS[690].VALUE := 0.0;
   STATUS[690].TRIGVALUE := 0.0;
   STATUS[690].EXT.AlarmWarnUnAck := FALSE;
   STATUS[690].EXT.AckRequired := FALSE;
   STATUS[690].EXT.Maintanence := FALSE;
   STATUS[690].EXT.Operation := FALSE;
   STATUS[690].EXT.Forced := FALSE;
   STATUS[690].EXT.BIT29 := FALSE;
   STATUS[690].EXT.BIT30 := FALSE;
   STATUS[690].EXT.BIT31 := FALSE;
   STATUS[690].EXT.ModeBit1 := FALSE;
   STATUS[690].EXT.ModeBit2 := FALSE;
   STATUS[690].EXT.ModeBit3 := FALSE;
   STATUS[690].EXT.BIT19 := FALSE;
   STATUS[690].EXT.BIT20 := FALSE;
   STATUS[690].EXT.AlarmSuppressed := FALSE;
   STATUS[690].EXT.AlarmPrsent := FALSE;
   STATUS[690].EXT.AlarmFailUnAck := FALSE;
   STATUS[690].Status := 0;
   STATUS[690].TimeStamp := 16#0000;
   STATUS[691].VALUE := 0.0;
   STATUS[691].TRIGVALUE := 0.0;
   STATUS[691].EXT.AlarmWarnUnAck := FALSE;
   STATUS[691].EXT.AckRequired := FALSE;
   STATUS[691].EXT.Maintanence := FALSE;
   STATUS[691].EXT.Operation := FALSE;
   STATUS[691].EXT.Forced := FALSE;
   STATUS[691].EXT.BIT29 := FALSE;
   STATUS[691].EXT.BIT30 := FALSE;
   STATUS[691].EXT.BIT31 := FALSE;
   STATUS[691].EXT.ModeBit1 := FALSE;
   STATUS[691].EXT.ModeBit2 := FALSE;
   STATUS[691].EXT.ModeBit3 := FALSE;
   STATUS[691].EXT.BIT19 := FALSE;
   STATUS[691].EXT.BIT20 := FALSE;
   STATUS[691].EXT.AlarmSuppressed := FALSE;
   STATUS[691].EXT.AlarmPrsent := FALSE;
   STATUS[691].EXT.AlarmFailUnAck := FALSE;
   STATUS[691].Status := 0;
   STATUS[691].TimeStamp := 16#0000;
   STATUS[692].VALUE := 0.0;
   STATUS[692].TRIGVALUE := 0.0;
   STATUS[692].EXT.AlarmWarnUnAck := FALSE;
   STATUS[692].EXT.AckRequired := FALSE;
   STATUS[692].EXT.Maintanence := FALSE;
   STATUS[692].EXT.Operation := FALSE;
   STATUS[692].EXT.Forced := FALSE;
   STATUS[692].EXT.BIT29 := FALSE;
   STATUS[692].EXT.BIT30 := FALSE;
   STATUS[692].EXT.BIT31 := FALSE;
   STATUS[692].EXT.ModeBit1 := FALSE;
   STATUS[692].EXT.ModeBit2 := FALSE;
   STATUS[692].EXT.ModeBit3 := FALSE;
   STATUS[692].EXT.BIT19 := FALSE;
   STATUS[692].EXT.BIT20 := FALSE;
   STATUS[692].EXT.AlarmSuppressed := FALSE;
   STATUS[692].EXT.AlarmPrsent := FALSE;
   STATUS[692].EXT.AlarmFailUnAck := FALSE;
   STATUS[692].Status := 0;
   STATUS[692].TimeStamp := 16#0000;
   STATUS[693].VALUE := 0.0;
   STATUS[693].TRIGVALUE := 0.0;
   STATUS[693].EXT.AlarmWarnUnAck := FALSE;
   STATUS[693].EXT.AckRequired := FALSE;
   STATUS[693].EXT.Maintanence := FALSE;
   STATUS[693].EXT.Operation := FALSE;
   STATUS[693].EXT.Forced := FALSE;
   STATUS[693].EXT.BIT29 := FALSE;
   STATUS[693].EXT.BIT30 := FALSE;
   STATUS[693].EXT.BIT31 := FALSE;
   STATUS[693].EXT.ModeBit1 := FALSE;
   STATUS[693].EXT.ModeBit2 := FALSE;
   STATUS[693].EXT.ModeBit3 := FALSE;
   STATUS[693].EXT.BIT19 := FALSE;
   STATUS[693].EXT.BIT20 := FALSE;
   STATUS[693].EXT.AlarmSuppressed := FALSE;
   STATUS[693].EXT.AlarmPrsent := FALSE;
   STATUS[693].EXT.AlarmFailUnAck := FALSE;
   STATUS[693].Status := 0;
   STATUS[693].TimeStamp := 16#0000;
   STATUS[694].VALUE := 0.0;
   STATUS[694].TRIGVALUE := 0.0;
   STATUS[694].EXT.AlarmWarnUnAck := FALSE;
   STATUS[694].EXT.AckRequired := FALSE;
   STATUS[694].EXT.Maintanence := FALSE;
   STATUS[694].EXT.Operation := FALSE;
   STATUS[694].EXT.Forced := FALSE;
   STATUS[694].EXT.BIT29 := FALSE;
   STATUS[694].EXT.BIT30 := FALSE;
   STATUS[694].EXT.BIT31 := FALSE;
   STATUS[694].EXT.ModeBit1 := FALSE;
   STATUS[694].EXT.ModeBit2 := FALSE;
   STATUS[694].EXT.ModeBit3 := FALSE;
   STATUS[694].EXT.BIT19 := FALSE;
   STATUS[694].EXT.BIT20 := FALSE;
   STATUS[694].EXT.AlarmSuppressed := FALSE;
   STATUS[694].EXT.AlarmPrsent := FALSE;
   STATUS[694].EXT.AlarmFailUnAck := FALSE;
   STATUS[694].Status := 0;
   STATUS[694].TimeStamp := 16#0000;
   STATUS[695].VALUE := 0.0;
   STATUS[695].TRIGVALUE := 0.0;
   STATUS[695].EXT.AlarmWarnUnAck := FALSE;
   STATUS[695].EXT.AckRequired := FALSE;
   STATUS[695].EXT.Maintanence := FALSE;
   STATUS[695].EXT.Operation := FALSE;
   STATUS[695].EXT.Forced := FALSE;
   STATUS[695].EXT.BIT29 := FALSE;
   STATUS[695].EXT.BIT30 := FALSE;
   STATUS[695].EXT.BIT31 := FALSE;
   STATUS[695].EXT.ModeBit1 := FALSE;
   STATUS[695].EXT.ModeBit2 := FALSE;
   STATUS[695].EXT.ModeBit3 := FALSE;
   STATUS[695].EXT.BIT19 := FALSE;
   STATUS[695].EXT.BIT20 := FALSE;
   STATUS[695].EXT.AlarmSuppressed := FALSE;
   STATUS[695].EXT.AlarmPrsent := FALSE;
   STATUS[695].EXT.AlarmFailUnAck := FALSE;
   STATUS[695].Status := 0;
   STATUS[695].TimeStamp := 16#0000;
   STATUS[696].VALUE := 0.0;
   STATUS[696].TRIGVALUE := 0.0;
   STATUS[696].EXT.AlarmWarnUnAck := FALSE;
   STATUS[696].EXT.AckRequired := FALSE;
   STATUS[696].EXT.Maintanence := FALSE;
   STATUS[696].EXT.Operation := FALSE;
   STATUS[696].EXT.Forced := FALSE;
   STATUS[696].EXT.BIT29 := FALSE;
   STATUS[696].EXT.BIT30 := FALSE;
   STATUS[696].EXT.BIT31 := FALSE;
   STATUS[696].EXT.ModeBit1 := FALSE;
   STATUS[696].EXT.ModeBit2 := FALSE;
   STATUS[696].EXT.ModeBit3 := FALSE;
   STATUS[696].EXT.BIT19 := FALSE;
   STATUS[696].EXT.BIT20 := FALSE;
   STATUS[696].EXT.AlarmSuppressed := FALSE;
   STATUS[696].EXT.AlarmPrsent := FALSE;
   STATUS[696].EXT.AlarmFailUnAck := FALSE;
   STATUS[696].Status := 0;
   STATUS[696].TimeStamp := 16#0000;
   STATUS[697].VALUE := 0.0;
   STATUS[697].TRIGVALUE := 0.0;
   STATUS[697].EXT.AlarmWarnUnAck := FALSE;
   STATUS[697].EXT.AckRequired := FALSE;
   STATUS[697].EXT.Maintanence := FALSE;
   STATUS[697].EXT.Operation := FALSE;
   STATUS[697].EXT.Forced := FALSE;
   STATUS[697].EXT.BIT29 := FALSE;
   STATUS[697].EXT.BIT30 := FALSE;
   STATUS[697].EXT.BIT31 := FALSE;
   STATUS[697].EXT.ModeBit1 := FALSE;
   STATUS[697].EXT.ModeBit2 := FALSE;
   STATUS[697].EXT.ModeBit3 := FALSE;
   STATUS[697].EXT.BIT19 := FALSE;
   STATUS[697].EXT.BIT20 := FALSE;
   STATUS[697].EXT.AlarmSuppressed := FALSE;
   STATUS[697].EXT.AlarmPrsent := FALSE;
   STATUS[697].EXT.AlarmFailUnAck := FALSE;
   STATUS[697].Status := 0;
   STATUS[697].TimeStamp := 16#0000;
   STATUS[698].VALUE := 0.0;
   STATUS[698].TRIGVALUE := 0.0;
   STATUS[698].EXT.AlarmWarnUnAck := FALSE;
   STATUS[698].EXT.AckRequired := FALSE;
   STATUS[698].EXT.Maintanence := FALSE;
   STATUS[698].EXT.Operation := FALSE;
   STATUS[698].EXT.Forced := FALSE;
   STATUS[698].EXT.BIT29 := FALSE;
   STATUS[698].EXT.BIT30 := FALSE;
   STATUS[698].EXT.BIT31 := FALSE;
   STATUS[698].EXT.ModeBit1 := FALSE;
   STATUS[698].EXT.ModeBit2 := FALSE;
   STATUS[698].EXT.ModeBit3 := FALSE;
   STATUS[698].EXT.BIT19 := FALSE;
   STATUS[698].EXT.BIT20 := FALSE;
   STATUS[698].EXT.AlarmSuppressed := FALSE;
   STATUS[698].EXT.AlarmPrsent := FALSE;
   STATUS[698].EXT.AlarmFailUnAck := FALSE;
   STATUS[698].Status := 0;
   STATUS[698].TimeStamp := 16#0000;
   STATUS[699].VALUE := 0.0;
   STATUS[699].TRIGVALUE := 0.0;
   STATUS[699].EXT.AlarmWarnUnAck := FALSE;
   STATUS[699].EXT.AckRequired := FALSE;
   STATUS[699].EXT.Maintanence := FALSE;
   STATUS[699].EXT.Operation := FALSE;
   STATUS[699].EXT.Forced := FALSE;
   STATUS[699].EXT.BIT29 := FALSE;
   STATUS[699].EXT.BIT30 := FALSE;
   STATUS[699].EXT.BIT31 := FALSE;
   STATUS[699].EXT.ModeBit1 := FALSE;
   STATUS[699].EXT.ModeBit2 := FALSE;
   STATUS[699].EXT.ModeBit3 := FALSE;
   STATUS[699].EXT.BIT19 := FALSE;
   STATUS[699].EXT.BIT20 := FALSE;
   STATUS[699].EXT.AlarmSuppressed := FALSE;
   STATUS[699].EXT.AlarmPrsent := FALSE;
   STATUS[699].EXT.AlarmFailUnAck := FALSE;
   STATUS[699].Status := 0;
   STATUS[699].TimeStamp := 16#0000;
   STATUS[700].VALUE := 0.0;
   STATUS[700].TRIGVALUE := 0.0;
   STATUS[700].EXT.AlarmWarnUnAck := FALSE;
   STATUS[700].EXT.AckRequired := FALSE;
   STATUS[700].EXT.Maintanence := FALSE;
   STATUS[700].EXT.Operation := FALSE;
   STATUS[700].EXT.Forced := FALSE;
   STATUS[700].EXT.BIT29 := FALSE;
   STATUS[700].EXT.BIT30 := FALSE;
   STATUS[700].EXT.BIT31 := FALSE;
   STATUS[700].EXT.ModeBit1 := FALSE;
   STATUS[700].EXT.ModeBit2 := FALSE;
   STATUS[700].EXT.ModeBit3 := FALSE;
   STATUS[700].EXT.BIT19 := FALSE;
   STATUS[700].EXT.BIT20 := FALSE;
   STATUS[700].EXT.AlarmSuppressed := FALSE;
   STATUS[700].EXT.AlarmPrsent := FALSE;
   STATUS[700].EXT.AlarmFailUnAck := FALSE;
   STATUS[700].Status := 0;
   STATUS[700].TimeStamp := 16#0000;
   STATUS[701].VALUE := 0.0;
   STATUS[701].TRIGVALUE := 0.0;
   STATUS[701].EXT.AlarmWarnUnAck := FALSE;
   STATUS[701].EXT.AckRequired := FALSE;
   STATUS[701].EXT.Maintanence := FALSE;
   STATUS[701].EXT.Operation := FALSE;
   STATUS[701].EXT.Forced := FALSE;
   STATUS[701].EXT.BIT29 := FALSE;
   STATUS[701].EXT.BIT30 := FALSE;
   STATUS[701].EXT.BIT31 := FALSE;
   STATUS[701].EXT.ModeBit1 := FALSE;
   STATUS[701].EXT.ModeBit2 := FALSE;
   STATUS[701].EXT.ModeBit3 := FALSE;
   STATUS[701].EXT.BIT19 := FALSE;
   STATUS[701].EXT.BIT20 := FALSE;
   STATUS[701].EXT.AlarmSuppressed := FALSE;
   STATUS[701].EXT.AlarmPrsent := FALSE;
   STATUS[701].EXT.AlarmFailUnAck := FALSE;
   STATUS[701].Status := 0;
   STATUS[701].TimeStamp := 16#0000;
   STATUS[702].VALUE := 0.0;
   STATUS[702].TRIGVALUE := 0.0;
   STATUS[702].EXT.AlarmWarnUnAck := FALSE;
   STATUS[702].EXT.AckRequired := FALSE;
   STATUS[702].EXT.Maintanence := FALSE;
   STATUS[702].EXT.Operation := FALSE;
   STATUS[702].EXT.Forced := FALSE;
   STATUS[702].EXT.BIT29 := FALSE;
   STATUS[702].EXT.BIT30 := FALSE;
   STATUS[702].EXT.BIT31 := FALSE;
   STATUS[702].EXT.ModeBit1 := FALSE;
   STATUS[702].EXT.ModeBit2 := FALSE;
   STATUS[702].EXT.ModeBit3 := FALSE;
   STATUS[702].EXT.BIT19 := FALSE;
   STATUS[702].EXT.BIT20 := FALSE;
   STATUS[702].EXT.AlarmSuppressed := FALSE;
   STATUS[702].EXT.AlarmPrsent := FALSE;
   STATUS[702].EXT.AlarmFailUnAck := FALSE;
   STATUS[702].Status := 0;
   STATUS[702].TimeStamp := 16#0000;
   STATUS[703].VALUE := 0.0;
   STATUS[703].TRIGVALUE := 0.0;
   STATUS[703].EXT.AlarmWarnUnAck := FALSE;
   STATUS[703].EXT.AckRequired := FALSE;
   STATUS[703].EXT.Maintanence := FALSE;
   STATUS[703].EXT.Operation := FALSE;
   STATUS[703].EXT.Forced := FALSE;
   STATUS[703].EXT.BIT29 := FALSE;
   STATUS[703].EXT.BIT30 := FALSE;
   STATUS[703].EXT.BIT31 := FALSE;
   STATUS[703].EXT.ModeBit1 := FALSE;
   STATUS[703].EXT.ModeBit2 := FALSE;
   STATUS[703].EXT.ModeBit3 := FALSE;
   STATUS[703].EXT.BIT19 := FALSE;
   STATUS[703].EXT.BIT20 := FALSE;
   STATUS[703].EXT.AlarmSuppressed := FALSE;
   STATUS[703].EXT.AlarmPrsent := FALSE;
   STATUS[703].EXT.AlarmFailUnAck := FALSE;
   STATUS[703].Status := 0;
   STATUS[703].TimeStamp := 16#0000;
   STATUS[704].VALUE := 0.0;
   STATUS[704].TRIGVALUE := 0.0;
   STATUS[704].EXT.AlarmWarnUnAck := FALSE;
   STATUS[704].EXT.AckRequired := FALSE;
   STATUS[704].EXT.Maintanence := FALSE;
   STATUS[704].EXT.Operation := FALSE;
   STATUS[704].EXT.Forced := FALSE;
   STATUS[704].EXT.BIT29 := FALSE;
   STATUS[704].EXT.BIT30 := FALSE;
   STATUS[704].EXT.BIT31 := FALSE;
   STATUS[704].EXT.ModeBit1 := FALSE;
   STATUS[704].EXT.ModeBit2 := FALSE;
   STATUS[704].EXT.ModeBit3 := FALSE;
   STATUS[704].EXT.BIT19 := FALSE;
   STATUS[704].EXT.BIT20 := FALSE;
   STATUS[704].EXT.AlarmSuppressed := FALSE;
   STATUS[704].EXT.AlarmPrsent := FALSE;
   STATUS[704].EXT.AlarmFailUnAck := FALSE;
   STATUS[704].Status := 0;
   STATUS[704].TimeStamp := 16#0000;
   STATUS[705].VALUE := 0.0;
   STATUS[705].TRIGVALUE := 0.0;
   STATUS[705].EXT.AlarmWarnUnAck := FALSE;
   STATUS[705].EXT.AckRequired := FALSE;
   STATUS[705].EXT.Maintanence := FALSE;
   STATUS[705].EXT.Operation := FALSE;
   STATUS[705].EXT.Forced := FALSE;
   STATUS[705].EXT.BIT29 := FALSE;
   STATUS[705].EXT.BIT30 := FALSE;
   STATUS[705].EXT.BIT31 := FALSE;
   STATUS[705].EXT.ModeBit1 := FALSE;
   STATUS[705].EXT.ModeBit2 := FALSE;
   STATUS[705].EXT.ModeBit3 := FALSE;
   STATUS[705].EXT.BIT19 := FALSE;
   STATUS[705].EXT.BIT20 := FALSE;
   STATUS[705].EXT.AlarmSuppressed := FALSE;
   STATUS[705].EXT.AlarmPrsent := FALSE;
   STATUS[705].EXT.AlarmFailUnAck := FALSE;
   STATUS[705].Status := 0;
   STATUS[705].TimeStamp := 16#0000;
   STATUS[706].VALUE := 0.0;
   STATUS[706].TRIGVALUE := 0.0;
   STATUS[706].EXT.AlarmWarnUnAck := FALSE;
   STATUS[706].EXT.AckRequired := FALSE;
   STATUS[706].EXT.Maintanence := FALSE;
   STATUS[706].EXT.Operation := FALSE;
   STATUS[706].EXT.Forced := FALSE;
   STATUS[706].EXT.BIT29 := FALSE;
   STATUS[706].EXT.BIT30 := FALSE;
   STATUS[706].EXT.BIT31 := FALSE;
   STATUS[706].EXT.ModeBit1 := FALSE;
   STATUS[706].EXT.ModeBit2 := FALSE;
   STATUS[706].EXT.ModeBit3 := FALSE;
   STATUS[706].EXT.BIT19 := FALSE;
   STATUS[706].EXT.BIT20 := FALSE;
   STATUS[706].EXT.AlarmSuppressed := FALSE;
   STATUS[706].EXT.AlarmPrsent := FALSE;
   STATUS[706].EXT.AlarmFailUnAck := FALSE;
   STATUS[706].Status := 0;
   STATUS[706].TimeStamp := 16#0000;
   STATUS[707].VALUE := 0.0;
   STATUS[707].TRIGVALUE := 0.0;
   STATUS[707].EXT.AlarmWarnUnAck := FALSE;
   STATUS[707].EXT.AckRequired := FALSE;
   STATUS[707].EXT.Maintanence := FALSE;
   STATUS[707].EXT.Operation := FALSE;
   STATUS[707].EXT.Forced := FALSE;
   STATUS[707].EXT.BIT29 := FALSE;
   STATUS[707].EXT.BIT30 := FALSE;
   STATUS[707].EXT.BIT31 := FALSE;
   STATUS[707].EXT.ModeBit1 := FALSE;
   STATUS[707].EXT.ModeBit2 := FALSE;
   STATUS[707].EXT.ModeBit3 := FALSE;
   STATUS[707].EXT.BIT19 := FALSE;
   STATUS[707].EXT.BIT20 := FALSE;
   STATUS[707].EXT.AlarmSuppressed := FALSE;
   STATUS[707].EXT.AlarmPrsent := FALSE;
   STATUS[707].EXT.AlarmFailUnAck := FALSE;
   STATUS[707].Status := 0;
   STATUS[707].TimeStamp := 16#0000;
   STATUS[708].VALUE := 0.0;
   STATUS[708].TRIGVALUE := 0.0;
   STATUS[708].EXT.AlarmWarnUnAck := FALSE;
   STATUS[708].EXT.AckRequired := FALSE;
   STATUS[708].EXT.Maintanence := FALSE;
   STATUS[708].EXT.Operation := FALSE;
   STATUS[708].EXT.Forced := FALSE;
   STATUS[708].EXT.BIT29 := FALSE;
   STATUS[708].EXT.BIT30 := FALSE;
   STATUS[708].EXT.BIT31 := FALSE;
   STATUS[708].EXT.ModeBit1 := FALSE;
   STATUS[708].EXT.ModeBit2 := FALSE;
   STATUS[708].EXT.ModeBit3 := FALSE;
   STATUS[708].EXT.BIT19 := FALSE;
   STATUS[708].EXT.BIT20 := FALSE;
   STATUS[708].EXT.AlarmSuppressed := FALSE;
   STATUS[708].EXT.AlarmPrsent := FALSE;
   STATUS[708].EXT.AlarmFailUnAck := FALSE;
   STATUS[708].Status := 0;
   STATUS[708].TimeStamp := 16#0000;
   STATUS[709].VALUE := 0.0;
   STATUS[709].TRIGVALUE := 0.0;
   STATUS[709].EXT.AlarmWarnUnAck := FALSE;
   STATUS[709].EXT.AckRequired := FALSE;
   STATUS[709].EXT.Maintanence := FALSE;
   STATUS[709].EXT.Operation := FALSE;
   STATUS[709].EXT.Forced := FALSE;
   STATUS[709].EXT.BIT29 := FALSE;
   STATUS[709].EXT.BIT30 := FALSE;
   STATUS[709].EXT.BIT31 := FALSE;
   STATUS[709].EXT.ModeBit1 := FALSE;
   STATUS[709].EXT.ModeBit2 := FALSE;
   STATUS[709].EXT.ModeBit3 := FALSE;
   STATUS[709].EXT.BIT19 := FALSE;
   STATUS[709].EXT.BIT20 := FALSE;
   STATUS[709].EXT.AlarmSuppressed := FALSE;
   STATUS[709].EXT.AlarmPrsent := FALSE;
   STATUS[709].EXT.AlarmFailUnAck := FALSE;
   STATUS[709].Status := 0;
   STATUS[709].TimeStamp := 16#0000;
   STATUS[710].VALUE := 0.0;
   STATUS[710].TRIGVALUE := 0.0;
   STATUS[710].EXT.AlarmWarnUnAck := FALSE;
   STATUS[710].EXT.AckRequired := FALSE;
   STATUS[710].EXT.Maintanence := FALSE;
   STATUS[710].EXT.Operation := FALSE;
   STATUS[710].EXT.Forced := FALSE;
   STATUS[710].EXT.BIT29 := FALSE;
   STATUS[710].EXT.BIT30 := FALSE;
   STATUS[710].EXT.BIT31 := FALSE;
   STATUS[710].EXT.ModeBit1 := FALSE;
   STATUS[710].EXT.ModeBit2 := FALSE;
   STATUS[710].EXT.ModeBit3 := FALSE;
   STATUS[710].EXT.BIT19 := FALSE;
   STATUS[710].EXT.BIT20 := FALSE;
   STATUS[710].EXT.AlarmSuppressed := FALSE;
   STATUS[710].EXT.AlarmPrsent := FALSE;
   STATUS[710].EXT.AlarmFailUnAck := FALSE;
   STATUS[710].Status := 0;
   STATUS[710].TimeStamp := 16#0000;
   STATUS[711].VALUE := 0.0;
   STATUS[711].TRIGVALUE := 0.0;
   STATUS[711].EXT.AlarmWarnUnAck := FALSE;
   STATUS[711].EXT.AckRequired := FALSE;
   STATUS[711].EXT.Maintanence := FALSE;
   STATUS[711].EXT.Operation := FALSE;
   STATUS[711].EXT.Forced := FALSE;
   STATUS[711].EXT.BIT29 := FALSE;
   STATUS[711].EXT.BIT30 := FALSE;
   STATUS[711].EXT.BIT31 := FALSE;
   STATUS[711].EXT.ModeBit1 := FALSE;
   STATUS[711].EXT.ModeBit2 := FALSE;
   STATUS[711].EXT.ModeBit3 := FALSE;
   STATUS[711].EXT.BIT19 := FALSE;
   STATUS[711].EXT.BIT20 := FALSE;
   STATUS[711].EXT.AlarmSuppressed := FALSE;
   STATUS[711].EXT.AlarmPrsent := FALSE;
   STATUS[711].EXT.AlarmFailUnAck := FALSE;
   STATUS[711].Status := 0;
   STATUS[711].TimeStamp := 16#0000;
   STATUS[712].VALUE := 0.0;
   STATUS[712].TRIGVALUE := 0.0;
   STATUS[712].EXT.AlarmWarnUnAck := FALSE;
   STATUS[712].EXT.AckRequired := FALSE;
   STATUS[712].EXT.Maintanence := FALSE;
   STATUS[712].EXT.Operation := FALSE;
   STATUS[712].EXT.Forced := FALSE;
   STATUS[712].EXT.BIT29 := FALSE;
   STATUS[712].EXT.BIT30 := FALSE;
   STATUS[712].EXT.BIT31 := FALSE;
   STATUS[712].EXT.ModeBit1 := FALSE;
   STATUS[712].EXT.ModeBit2 := FALSE;
   STATUS[712].EXT.ModeBit3 := FALSE;
   STATUS[712].EXT.BIT19 := FALSE;
   STATUS[712].EXT.BIT20 := FALSE;
   STATUS[712].EXT.AlarmSuppressed := FALSE;
   STATUS[712].EXT.AlarmPrsent := FALSE;
   STATUS[712].EXT.AlarmFailUnAck := FALSE;
   STATUS[712].Status := 0;
   STATUS[712].TimeStamp := 16#0000;
   STATUS[713].VALUE := 0.0;
   STATUS[713].TRIGVALUE := 0.0;
   STATUS[713].EXT.AlarmWarnUnAck := FALSE;
   STATUS[713].EXT.AckRequired := FALSE;
   STATUS[713].EXT.Maintanence := FALSE;
   STATUS[713].EXT.Operation := FALSE;
   STATUS[713].EXT.Forced := FALSE;
   STATUS[713].EXT.BIT29 := FALSE;
   STATUS[713].EXT.BIT30 := FALSE;
   STATUS[713].EXT.BIT31 := FALSE;
   STATUS[713].EXT.ModeBit1 := FALSE;
   STATUS[713].EXT.ModeBit2 := FALSE;
   STATUS[713].EXT.ModeBit3 := FALSE;
   STATUS[713].EXT.BIT19 := FALSE;
   STATUS[713].EXT.BIT20 := FALSE;
   STATUS[713].EXT.AlarmSuppressed := FALSE;
   STATUS[713].EXT.AlarmPrsent := FALSE;
   STATUS[713].EXT.AlarmFailUnAck := FALSE;
   STATUS[713].Status := 0;
   STATUS[713].TimeStamp := 16#0000;
   STATUS[714].VALUE := 0.0;
   STATUS[714].TRIGVALUE := 0.0;
   STATUS[714].EXT.AlarmWarnUnAck := FALSE;
   STATUS[714].EXT.AckRequired := FALSE;
   STATUS[714].EXT.Maintanence := FALSE;
   STATUS[714].EXT.Operation := FALSE;
   STATUS[714].EXT.Forced := FALSE;
   STATUS[714].EXT.BIT29 := FALSE;
   STATUS[714].EXT.BIT30 := FALSE;
   STATUS[714].EXT.BIT31 := FALSE;
   STATUS[714].EXT.ModeBit1 := FALSE;
   STATUS[714].EXT.ModeBit2 := FALSE;
   STATUS[714].EXT.ModeBit3 := FALSE;
   STATUS[714].EXT.BIT19 := FALSE;
   STATUS[714].EXT.BIT20 := FALSE;
   STATUS[714].EXT.AlarmSuppressed := FALSE;
   STATUS[714].EXT.AlarmPrsent := FALSE;
   STATUS[714].EXT.AlarmFailUnAck := FALSE;
   STATUS[714].Status := 0;
   STATUS[714].TimeStamp := 16#0000;
   STATUS[715].VALUE := 0.0;
   STATUS[715].TRIGVALUE := 0.0;
   STATUS[715].EXT.AlarmWarnUnAck := FALSE;
   STATUS[715].EXT.AckRequired := FALSE;
   STATUS[715].EXT.Maintanence := FALSE;
   STATUS[715].EXT.Operation := FALSE;
   STATUS[715].EXT.Forced := FALSE;
   STATUS[715].EXT.BIT29 := FALSE;
   STATUS[715].EXT.BIT30 := FALSE;
   STATUS[715].EXT.BIT31 := FALSE;
   STATUS[715].EXT.ModeBit1 := FALSE;
   STATUS[715].EXT.ModeBit2 := FALSE;
   STATUS[715].EXT.ModeBit3 := FALSE;
   STATUS[715].EXT.BIT19 := FALSE;
   STATUS[715].EXT.BIT20 := FALSE;
   STATUS[715].EXT.AlarmSuppressed := FALSE;
   STATUS[715].EXT.AlarmPrsent := FALSE;
   STATUS[715].EXT.AlarmFailUnAck := FALSE;
   STATUS[715].Status := 0;
   STATUS[715].TimeStamp := 16#0000;
   STATUS[716].VALUE := 0.0;
   STATUS[716].TRIGVALUE := 0.0;
   STATUS[716].EXT.AlarmWarnUnAck := FALSE;
   STATUS[716].EXT.AckRequired := FALSE;
   STATUS[716].EXT.Maintanence := FALSE;
   STATUS[716].EXT.Operation := FALSE;
   STATUS[716].EXT.Forced := FALSE;
   STATUS[716].EXT.BIT29 := FALSE;
   STATUS[716].EXT.BIT30 := FALSE;
   STATUS[716].EXT.BIT31 := FALSE;
   STATUS[716].EXT.ModeBit1 := FALSE;
   STATUS[716].EXT.ModeBit2 := FALSE;
   STATUS[716].EXT.ModeBit3 := FALSE;
   STATUS[716].EXT.BIT19 := FALSE;
   STATUS[716].EXT.BIT20 := FALSE;
   STATUS[716].EXT.AlarmSuppressed := FALSE;
   STATUS[716].EXT.AlarmPrsent := FALSE;
   STATUS[716].EXT.AlarmFailUnAck := FALSE;
   STATUS[716].Status := 0;
   STATUS[716].TimeStamp := 16#0000;
   STATUS[717].VALUE := 0.0;
   STATUS[717].TRIGVALUE := 0.0;
   STATUS[717].EXT.AlarmWarnUnAck := FALSE;
   STATUS[717].EXT.AckRequired := FALSE;
   STATUS[717].EXT.Maintanence := FALSE;
   STATUS[717].EXT.Operation := FALSE;
   STATUS[717].EXT.Forced := FALSE;
   STATUS[717].EXT.BIT29 := FALSE;
   STATUS[717].EXT.BIT30 := FALSE;
   STATUS[717].EXT.BIT31 := FALSE;
   STATUS[717].EXT.ModeBit1 := FALSE;
   STATUS[717].EXT.ModeBit2 := FALSE;
   STATUS[717].EXT.ModeBit3 := FALSE;
   STATUS[717].EXT.BIT19 := FALSE;
   STATUS[717].EXT.BIT20 := FALSE;
   STATUS[717].EXT.AlarmSuppressed := FALSE;
   STATUS[717].EXT.AlarmPrsent := FALSE;
   STATUS[717].EXT.AlarmFailUnAck := FALSE;
   STATUS[717].Status := 0;
   STATUS[717].TimeStamp := 16#0000;
   STATUS[718].VALUE := 0.0;
   STATUS[718].TRIGVALUE := 0.0;
   STATUS[718].EXT.AlarmWarnUnAck := FALSE;
   STATUS[718].EXT.AckRequired := FALSE;
   STATUS[718].EXT.Maintanence := FALSE;
   STATUS[718].EXT.Operation := FALSE;
   STATUS[718].EXT.Forced := FALSE;
   STATUS[718].EXT.BIT29 := FALSE;
   STATUS[718].EXT.BIT30 := FALSE;
   STATUS[718].EXT.BIT31 := FALSE;
   STATUS[718].EXT.ModeBit1 := FALSE;
   STATUS[718].EXT.ModeBit2 := FALSE;
   STATUS[718].EXT.ModeBit3 := FALSE;
   STATUS[718].EXT.BIT19 := FALSE;
   STATUS[718].EXT.BIT20 := FALSE;
   STATUS[718].EXT.AlarmSuppressed := FALSE;
   STATUS[718].EXT.AlarmPrsent := FALSE;
   STATUS[718].EXT.AlarmFailUnAck := FALSE;
   STATUS[718].Status := 0;
   STATUS[718].TimeStamp := 16#0000;
   STATUS[719].VALUE := 0.0;
   STATUS[719].TRIGVALUE := 0.0;
   STATUS[719].EXT.AlarmWarnUnAck := FALSE;
   STATUS[719].EXT.AckRequired := FALSE;
   STATUS[719].EXT.Maintanence := FALSE;
   STATUS[719].EXT.Operation := FALSE;
   STATUS[719].EXT.Forced := FALSE;
   STATUS[719].EXT.BIT29 := FALSE;
   STATUS[719].EXT.BIT30 := FALSE;
   STATUS[719].EXT.BIT31 := FALSE;
   STATUS[719].EXT.ModeBit1 := FALSE;
   STATUS[719].EXT.ModeBit2 := FALSE;
   STATUS[719].EXT.ModeBit3 := FALSE;
   STATUS[719].EXT.BIT19 := FALSE;
   STATUS[719].EXT.BIT20 := FALSE;
   STATUS[719].EXT.AlarmSuppressed := FALSE;
   STATUS[719].EXT.AlarmPrsent := FALSE;
   STATUS[719].EXT.AlarmFailUnAck := FALSE;
   STATUS[719].Status := 0;
   STATUS[719].TimeStamp := 16#0000;
   STATUS[720].VALUE := 0.0;
   STATUS[720].TRIGVALUE := 0.0;
   STATUS[720].EXT.AlarmWarnUnAck := FALSE;
   STATUS[720].EXT.AckRequired := FALSE;
   STATUS[720].EXT.Maintanence := FALSE;
   STATUS[720].EXT.Operation := FALSE;
   STATUS[720].EXT.Forced := FALSE;
   STATUS[720].EXT.BIT29 := FALSE;
   STATUS[720].EXT.BIT30 := FALSE;
   STATUS[720].EXT.BIT31 := FALSE;
   STATUS[720].EXT.ModeBit1 := FALSE;
   STATUS[720].EXT.ModeBit2 := FALSE;
   STATUS[720].EXT.ModeBit3 := FALSE;
   STATUS[720].EXT.BIT19 := FALSE;
   STATUS[720].EXT.BIT20 := FALSE;
   STATUS[720].EXT.AlarmSuppressed := FALSE;
   STATUS[720].EXT.AlarmPrsent := FALSE;
   STATUS[720].EXT.AlarmFailUnAck := FALSE;
   STATUS[720].Status := 0;
   STATUS[720].TimeStamp := 16#0000;
   STATUS[721].VALUE := 0.0;
   STATUS[721].TRIGVALUE := 0.0;
   STATUS[721].EXT.AlarmWarnUnAck := FALSE;
   STATUS[721].EXT.AckRequired := FALSE;
   STATUS[721].EXT.Maintanence := FALSE;
   STATUS[721].EXT.Operation := FALSE;
   STATUS[721].EXT.Forced := FALSE;
   STATUS[721].EXT.BIT29 := FALSE;
   STATUS[721].EXT.BIT30 := FALSE;
   STATUS[721].EXT.BIT31 := FALSE;
   STATUS[721].EXT.ModeBit1 := FALSE;
   STATUS[721].EXT.ModeBit2 := FALSE;
   STATUS[721].EXT.ModeBit3 := FALSE;
   STATUS[721].EXT.BIT19 := FALSE;
   STATUS[721].EXT.BIT20 := FALSE;
   STATUS[721].EXT.AlarmSuppressed := FALSE;
   STATUS[721].EXT.AlarmPrsent := FALSE;
   STATUS[721].EXT.AlarmFailUnAck := FALSE;
   STATUS[721].Status := 0;
   STATUS[721].TimeStamp := 16#0000;
   STATUS[722].VALUE := 0.0;
   STATUS[722].TRIGVALUE := 0.0;
   STATUS[722].EXT.AlarmWarnUnAck := FALSE;
   STATUS[722].EXT.AckRequired := FALSE;
   STATUS[722].EXT.Maintanence := FALSE;
   STATUS[722].EXT.Operation := FALSE;
   STATUS[722].EXT.Forced := FALSE;
   STATUS[722].EXT.BIT29 := FALSE;
   STATUS[722].EXT.BIT30 := FALSE;
   STATUS[722].EXT.BIT31 := FALSE;
   STATUS[722].EXT.ModeBit1 := FALSE;
   STATUS[722].EXT.ModeBit2 := FALSE;
   STATUS[722].EXT.ModeBit3 := FALSE;
   STATUS[722].EXT.BIT19 := FALSE;
   STATUS[722].EXT.BIT20 := FALSE;
   STATUS[722].EXT.AlarmSuppressed := FALSE;
   STATUS[722].EXT.AlarmPrsent := FALSE;
   STATUS[722].EXT.AlarmFailUnAck := FALSE;
   STATUS[722].Status := 0;
   STATUS[722].TimeStamp := 16#0000;
   STATUS[723].VALUE := 0.0;
   STATUS[723].TRIGVALUE := 0.0;
   STATUS[723].EXT.AlarmWarnUnAck := FALSE;
   STATUS[723].EXT.AckRequired := FALSE;
   STATUS[723].EXT.Maintanence := FALSE;
   STATUS[723].EXT.Operation := FALSE;
   STATUS[723].EXT.Forced := FALSE;
   STATUS[723].EXT.BIT29 := FALSE;
   STATUS[723].EXT.BIT30 := FALSE;
   STATUS[723].EXT.BIT31 := FALSE;
   STATUS[723].EXT.ModeBit1 := FALSE;
   STATUS[723].EXT.ModeBit2 := FALSE;
   STATUS[723].EXT.ModeBit3 := FALSE;
   STATUS[723].EXT.BIT19 := FALSE;
   STATUS[723].EXT.BIT20 := FALSE;
   STATUS[723].EXT.AlarmSuppressed := FALSE;
   STATUS[723].EXT.AlarmPrsent := FALSE;
   STATUS[723].EXT.AlarmFailUnAck := FALSE;
   STATUS[723].Status := 0;
   STATUS[723].TimeStamp := 16#0000;
   STATUS[724].VALUE := 0.0;
   STATUS[724].TRIGVALUE := 0.0;
   STATUS[724].EXT.AlarmWarnUnAck := FALSE;
   STATUS[724].EXT.AckRequired := FALSE;
   STATUS[724].EXT.Maintanence := FALSE;
   STATUS[724].EXT.Operation := FALSE;
   STATUS[724].EXT.Forced := FALSE;
   STATUS[724].EXT.BIT29 := FALSE;
   STATUS[724].EXT.BIT30 := FALSE;
   STATUS[724].EXT.BIT31 := FALSE;
   STATUS[724].EXT.ModeBit1 := FALSE;
   STATUS[724].EXT.ModeBit2 := FALSE;
   STATUS[724].EXT.ModeBit3 := FALSE;
   STATUS[724].EXT.BIT19 := FALSE;
   STATUS[724].EXT.BIT20 := FALSE;
   STATUS[724].EXT.AlarmSuppressed := FALSE;
   STATUS[724].EXT.AlarmPrsent := FALSE;
   STATUS[724].EXT.AlarmFailUnAck := FALSE;
   STATUS[724].Status := 0;
   STATUS[724].TimeStamp := 16#0000;
   STATUS[725].VALUE := 0.0;
   STATUS[725].TRIGVALUE := 0.0;
   STATUS[725].EXT.AlarmWarnUnAck := FALSE;
   STATUS[725].EXT.AckRequired := FALSE;
   STATUS[725].EXT.Maintanence := FALSE;
   STATUS[725].EXT.Operation := FALSE;
   STATUS[725].EXT.Forced := FALSE;
   STATUS[725].EXT.BIT29 := FALSE;
   STATUS[725].EXT.BIT30 := FALSE;
   STATUS[725].EXT.BIT31 := FALSE;
   STATUS[725].EXT.ModeBit1 := FALSE;
   STATUS[725].EXT.ModeBit2 := FALSE;
   STATUS[725].EXT.ModeBit3 := FALSE;
   STATUS[725].EXT.BIT19 := FALSE;
   STATUS[725].EXT.BIT20 := FALSE;
   STATUS[725].EXT.AlarmSuppressed := FALSE;
   STATUS[725].EXT.AlarmPrsent := FALSE;
   STATUS[725].EXT.AlarmFailUnAck := FALSE;
   STATUS[725].Status := 0;
   STATUS[725].TimeStamp := 16#0000;
   STATUS[726].VALUE := 0.0;
   STATUS[726].TRIGVALUE := 0.0;
   STATUS[726].EXT.AlarmWarnUnAck := FALSE;
   STATUS[726].EXT.AckRequired := FALSE;
   STATUS[726].EXT.Maintanence := FALSE;
   STATUS[726].EXT.Operation := FALSE;
   STATUS[726].EXT.Forced := FALSE;
   STATUS[726].EXT.BIT29 := FALSE;
   STATUS[726].EXT.BIT30 := FALSE;
   STATUS[726].EXT.BIT31 := FALSE;
   STATUS[726].EXT.ModeBit1 := FALSE;
   STATUS[726].EXT.ModeBit2 := FALSE;
   STATUS[726].EXT.ModeBit3 := FALSE;
   STATUS[726].EXT.BIT19 := FALSE;
   STATUS[726].EXT.BIT20 := FALSE;
   STATUS[726].EXT.AlarmSuppressed := FALSE;
   STATUS[726].EXT.AlarmPrsent := FALSE;
   STATUS[726].EXT.AlarmFailUnAck := FALSE;
   STATUS[726].Status := 0;
   STATUS[726].TimeStamp := 16#0000;
   STATUS[727].VALUE := 0.0;
   STATUS[727].TRIGVALUE := 0.0;
   STATUS[727].EXT.AlarmWarnUnAck := FALSE;
   STATUS[727].EXT.AckRequired := FALSE;
   STATUS[727].EXT.Maintanence := FALSE;
   STATUS[727].EXT.Operation := FALSE;
   STATUS[727].EXT.Forced := FALSE;
   STATUS[727].EXT.BIT29 := FALSE;
   STATUS[727].EXT.BIT30 := FALSE;
   STATUS[727].EXT.BIT31 := FALSE;
   STATUS[727].EXT.ModeBit1 := FALSE;
   STATUS[727].EXT.ModeBit2 := FALSE;
   STATUS[727].EXT.ModeBit3 := FALSE;
   STATUS[727].EXT.BIT19 := FALSE;
   STATUS[727].EXT.BIT20 := FALSE;
   STATUS[727].EXT.AlarmSuppressed := FALSE;
   STATUS[727].EXT.AlarmPrsent := FALSE;
   STATUS[727].EXT.AlarmFailUnAck := FALSE;
   STATUS[727].Status := 0;
   STATUS[727].TimeStamp := 16#0000;
   STATUS[728].VALUE := 0.0;
   STATUS[728].TRIGVALUE := 0.0;
   STATUS[728].EXT.AlarmWarnUnAck := FALSE;
   STATUS[728].EXT.AckRequired := FALSE;
   STATUS[728].EXT.Maintanence := FALSE;
   STATUS[728].EXT.Operation := FALSE;
   STATUS[728].EXT.Forced := FALSE;
   STATUS[728].EXT.BIT29 := FALSE;
   STATUS[728].EXT.BIT30 := FALSE;
   STATUS[728].EXT.BIT31 := FALSE;
   STATUS[728].EXT.ModeBit1 := FALSE;
   STATUS[728].EXT.ModeBit2 := FALSE;
   STATUS[728].EXT.ModeBit3 := FALSE;
   STATUS[728].EXT.BIT19 := FALSE;
   STATUS[728].EXT.BIT20 := FALSE;
   STATUS[728].EXT.AlarmSuppressed := FALSE;
   STATUS[728].EXT.AlarmPrsent := FALSE;
   STATUS[728].EXT.AlarmFailUnAck := FALSE;
   STATUS[728].Status := 0;
   STATUS[728].TimeStamp := 16#0000;
   STATUS[729].VALUE := 0.0;
   STATUS[729].TRIGVALUE := 0.0;
   STATUS[729].EXT.AlarmWarnUnAck := FALSE;
   STATUS[729].EXT.AckRequired := FALSE;
   STATUS[729].EXT.Maintanence := FALSE;
   STATUS[729].EXT.Operation := FALSE;
   STATUS[729].EXT.Forced := FALSE;
   STATUS[729].EXT.BIT29 := FALSE;
   STATUS[729].EXT.BIT30 := FALSE;
   STATUS[729].EXT.BIT31 := FALSE;
   STATUS[729].EXT.ModeBit1 := FALSE;
   STATUS[729].EXT.ModeBit2 := FALSE;
   STATUS[729].EXT.ModeBit3 := FALSE;
   STATUS[729].EXT.BIT19 := FALSE;
   STATUS[729].EXT.BIT20 := FALSE;
   STATUS[729].EXT.AlarmSuppressed := FALSE;
   STATUS[729].EXT.AlarmPrsent := FALSE;
   STATUS[729].EXT.AlarmFailUnAck := FALSE;
   STATUS[729].Status := 0;
   STATUS[729].TimeStamp := 16#0000;
   STATUS[730].VALUE := 0.0;
   STATUS[730].TRIGVALUE := 0.0;
   STATUS[730].EXT.AlarmWarnUnAck := FALSE;
   STATUS[730].EXT.AckRequired := FALSE;
   STATUS[730].EXT.Maintanence := FALSE;
   STATUS[730].EXT.Operation := FALSE;
   STATUS[730].EXT.Forced := FALSE;
   STATUS[730].EXT.BIT29 := FALSE;
   STATUS[730].EXT.BIT30 := FALSE;
   STATUS[730].EXT.BIT31 := FALSE;
   STATUS[730].EXT.ModeBit1 := FALSE;
   STATUS[730].EXT.ModeBit2 := FALSE;
   STATUS[730].EXT.ModeBit3 := FALSE;
   STATUS[730].EXT.BIT19 := FALSE;
   STATUS[730].EXT.BIT20 := FALSE;
   STATUS[730].EXT.AlarmSuppressed := FALSE;
   STATUS[730].EXT.AlarmPrsent := FALSE;
   STATUS[730].EXT.AlarmFailUnAck := FALSE;
   STATUS[730].Status := 0;
   STATUS[730].TimeStamp := 16#0000;
   STATUS[731].VALUE := 0.0;
   STATUS[731].TRIGVALUE := 0.0;
   STATUS[731].EXT.AlarmWarnUnAck := FALSE;
   STATUS[731].EXT.AckRequired := FALSE;
   STATUS[731].EXT.Maintanence := FALSE;
   STATUS[731].EXT.Operation := FALSE;
   STATUS[731].EXT.Forced := FALSE;
   STATUS[731].EXT.BIT29 := FALSE;
   STATUS[731].EXT.BIT30 := FALSE;
   STATUS[731].EXT.BIT31 := FALSE;
   STATUS[731].EXT.ModeBit1 := FALSE;
   STATUS[731].EXT.ModeBit2 := FALSE;
   STATUS[731].EXT.ModeBit3 := FALSE;
   STATUS[731].EXT.BIT19 := FALSE;
   STATUS[731].EXT.BIT20 := FALSE;
   STATUS[731].EXT.AlarmSuppressed := FALSE;
   STATUS[731].EXT.AlarmPrsent := FALSE;
   STATUS[731].EXT.AlarmFailUnAck := FALSE;
   STATUS[731].Status := 0;
   STATUS[731].TimeStamp := 16#0000;
   STATUS[732].VALUE := 0.0;
   STATUS[732].TRIGVALUE := 0.0;
   STATUS[732].EXT.AlarmWarnUnAck := FALSE;
   STATUS[732].EXT.AckRequired := FALSE;
   STATUS[732].EXT.Maintanence := FALSE;
   STATUS[732].EXT.Operation := FALSE;
   STATUS[732].EXT.Forced := FALSE;
   STATUS[732].EXT.BIT29 := FALSE;
   STATUS[732].EXT.BIT30 := FALSE;
   STATUS[732].EXT.BIT31 := FALSE;
   STATUS[732].EXT.ModeBit1 := FALSE;
   STATUS[732].EXT.ModeBit2 := FALSE;
   STATUS[732].EXT.ModeBit3 := FALSE;
   STATUS[732].EXT.BIT19 := FALSE;
   STATUS[732].EXT.BIT20 := FALSE;
   STATUS[732].EXT.AlarmSuppressed := FALSE;
   STATUS[732].EXT.AlarmPrsent := FALSE;
   STATUS[732].EXT.AlarmFailUnAck := FALSE;
   STATUS[732].Status := 0;
   STATUS[732].TimeStamp := 16#0000;
   STATUS[733].VALUE := 0.0;
   STATUS[733].TRIGVALUE := 0.0;
   STATUS[733].EXT.AlarmWarnUnAck := FALSE;
   STATUS[733].EXT.AckRequired := FALSE;
   STATUS[733].EXT.Maintanence := FALSE;
   STATUS[733].EXT.Operation := FALSE;
   STATUS[733].EXT.Forced := FALSE;
   STATUS[733].EXT.BIT29 := FALSE;
   STATUS[733].EXT.BIT30 := FALSE;
   STATUS[733].EXT.BIT31 := FALSE;
   STATUS[733].EXT.ModeBit1 := FALSE;
   STATUS[733].EXT.ModeBit2 := FALSE;
   STATUS[733].EXT.ModeBit3 := FALSE;
   STATUS[733].EXT.BIT19 := FALSE;
   STATUS[733].EXT.BIT20 := FALSE;
   STATUS[733].EXT.AlarmSuppressed := FALSE;
   STATUS[733].EXT.AlarmPrsent := FALSE;
   STATUS[733].EXT.AlarmFailUnAck := FALSE;
   STATUS[733].Status := 0;
   STATUS[733].TimeStamp := 16#0000;
   STATUS[734].VALUE := 0.0;
   STATUS[734].TRIGVALUE := 0.0;
   STATUS[734].EXT.AlarmWarnUnAck := FALSE;
   STATUS[734].EXT.AckRequired := FALSE;
   STATUS[734].EXT.Maintanence := FALSE;
   STATUS[734].EXT.Operation := FALSE;
   STATUS[734].EXT.Forced := FALSE;
   STATUS[734].EXT.BIT29 := FALSE;
   STATUS[734].EXT.BIT30 := FALSE;
   STATUS[734].EXT.BIT31 := FALSE;
   STATUS[734].EXT.ModeBit1 := FALSE;
   STATUS[734].EXT.ModeBit2 := FALSE;
   STATUS[734].EXT.ModeBit3 := FALSE;
   STATUS[734].EXT.BIT19 := FALSE;
   STATUS[734].EXT.BIT20 := FALSE;
   STATUS[734].EXT.AlarmSuppressed := FALSE;
   STATUS[734].EXT.AlarmPrsent := FALSE;
   STATUS[734].EXT.AlarmFailUnAck := FALSE;
   STATUS[734].Status := 0;
   STATUS[734].TimeStamp := 16#0000;
   STATUS[735].VALUE := 0.0;
   STATUS[735].TRIGVALUE := 0.0;
   STATUS[735].EXT.AlarmWarnUnAck := FALSE;
   STATUS[735].EXT.AckRequired := FALSE;
   STATUS[735].EXT.Maintanence := FALSE;
   STATUS[735].EXT.Operation := FALSE;
   STATUS[735].EXT.Forced := FALSE;
   STATUS[735].EXT.BIT29 := FALSE;
   STATUS[735].EXT.BIT30 := FALSE;
   STATUS[735].EXT.BIT31 := FALSE;
   STATUS[735].EXT.ModeBit1 := FALSE;
   STATUS[735].EXT.ModeBit2 := FALSE;
   STATUS[735].EXT.ModeBit3 := FALSE;
   STATUS[735].EXT.BIT19 := FALSE;
   STATUS[735].EXT.BIT20 := FALSE;
   STATUS[735].EXT.AlarmSuppressed := FALSE;
   STATUS[735].EXT.AlarmPrsent := FALSE;
   STATUS[735].EXT.AlarmFailUnAck := FALSE;
   STATUS[735].Status := 0;
   STATUS[735].TimeStamp := 16#0000;
   STATUS[736].VALUE := 0.0;
   STATUS[736].TRIGVALUE := 0.0;
   STATUS[736].EXT.AlarmWarnUnAck := FALSE;
   STATUS[736].EXT.AckRequired := FALSE;
   STATUS[736].EXT.Maintanence := FALSE;
   STATUS[736].EXT.Operation := FALSE;
   STATUS[736].EXT.Forced := FALSE;
   STATUS[736].EXT.BIT29 := FALSE;
   STATUS[736].EXT.BIT30 := FALSE;
   STATUS[736].EXT.BIT31 := FALSE;
   STATUS[736].EXT.ModeBit1 := FALSE;
   STATUS[736].EXT.ModeBit2 := FALSE;
   STATUS[736].EXT.ModeBit3 := FALSE;
   STATUS[736].EXT.BIT19 := FALSE;
   STATUS[736].EXT.BIT20 := FALSE;
   STATUS[736].EXT.AlarmSuppressed := FALSE;
   STATUS[736].EXT.AlarmPrsent := FALSE;
   STATUS[736].EXT.AlarmFailUnAck := FALSE;
   STATUS[736].Status := 0;
   STATUS[736].TimeStamp := 16#0000;
   STATUS[737].VALUE := 0.0;
   STATUS[737].TRIGVALUE := 0.0;
   STATUS[737].EXT.AlarmWarnUnAck := FALSE;
   STATUS[737].EXT.AckRequired := FALSE;
   STATUS[737].EXT.Maintanence := FALSE;
   STATUS[737].EXT.Operation := FALSE;
   STATUS[737].EXT.Forced := FALSE;
   STATUS[737].EXT.BIT29 := FALSE;
   STATUS[737].EXT.BIT30 := FALSE;
   STATUS[737].EXT.BIT31 := FALSE;
   STATUS[737].EXT.ModeBit1 := FALSE;
   STATUS[737].EXT.ModeBit2 := FALSE;
   STATUS[737].EXT.ModeBit3 := FALSE;
   STATUS[737].EXT.BIT19 := FALSE;
   STATUS[737].EXT.BIT20 := FALSE;
   STATUS[737].EXT.AlarmSuppressed := FALSE;
   STATUS[737].EXT.AlarmPrsent := FALSE;
   STATUS[737].EXT.AlarmFailUnAck := FALSE;
   STATUS[737].Status := 0;
   STATUS[737].TimeStamp := 16#0000;
   STATUS[738].VALUE := 0.0;
   STATUS[738].TRIGVALUE := 0.0;
   STATUS[738].EXT.AlarmWarnUnAck := FALSE;
   STATUS[738].EXT.AckRequired := FALSE;
   STATUS[738].EXT.Maintanence := FALSE;
   STATUS[738].EXT.Operation := FALSE;
   STATUS[738].EXT.Forced := FALSE;
   STATUS[738].EXT.BIT29 := FALSE;
   STATUS[738].EXT.BIT30 := FALSE;
   STATUS[738].EXT.BIT31 := FALSE;
   STATUS[738].EXT.ModeBit1 := FALSE;
   STATUS[738].EXT.ModeBit2 := FALSE;
   STATUS[738].EXT.ModeBit3 := FALSE;
   STATUS[738].EXT.BIT19 := FALSE;
   STATUS[738].EXT.BIT20 := FALSE;
   STATUS[738].EXT.AlarmSuppressed := FALSE;
   STATUS[738].EXT.AlarmPrsent := FALSE;
   STATUS[738].EXT.AlarmFailUnAck := FALSE;
   STATUS[738].Status := 0;
   STATUS[738].TimeStamp := 16#0000;
   STATUS[739].VALUE := 0.0;
   STATUS[739].TRIGVALUE := 0.0;
   STATUS[739].EXT.AlarmWarnUnAck := FALSE;
   STATUS[739].EXT.AckRequired := FALSE;
   STATUS[739].EXT.Maintanence := FALSE;
   STATUS[739].EXT.Operation := FALSE;
   STATUS[739].EXT.Forced := FALSE;
   STATUS[739].EXT.BIT29 := FALSE;
   STATUS[739].EXT.BIT30 := FALSE;
   STATUS[739].EXT.BIT31 := FALSE;
   STATUS[739].EXT.ModeBit1 := FALSE;
   STATUS[739].EXT.ModeBit2 := FALSE;
   STATUS[739].EXT.ModeBit3 := FALSE;
   STATUS[739].EXT.BIT19 := FALSE;
   STATUS[739].EXT.BIT20 := FALSE;
   STATUS[739].EXT.AlarmSuppressed := FALSE;
   STATUS[739].EXT.AlarmPrsent := FALSE;
   STATUS[739].EXT.AlarmFailUnAck := FALSE;
   STATUS[739].Status := 0;
   STATUS[739].TimeStamp := 16#0000;
   STATUS[740].VALUE := 0.0;
   STATUS[740].TRIGVALUE := 0.0;
   STATUS[740].EXT.AlarmWarnUnAck := FALSE;
   STATUS[740].EXT.AckRequired := FALSE;
   STATUS[740].EXT.Maintanence := FALSE;
   STATUS[740].EXT.Operation := FALSE;
   STATUS[740].EXT.Forced := FALSE;
   STATUS[740].EXT.BIT29 := FALSE;
   STATUS[740].EXT.BIT30 := FALSE;
   STATUS[740].EXT.BIT31 := FALSE;
   STATUS[740].EXT.ModeBit1 := FALSE;
   STATUS[740].EXT.ModeBit2 := FALSE;
   STATUS[740].EXT.ModeBit3 := FALSE;
   STATUS[740].EXT.BIT19 := FALSE;
   STATUS[740].EXT.BIT20 := FALSE;
   STATUS[740].EXT.AlarmSuppressed := FALSE;
   STATUS[740].EXT.AlarmPrsent := FALSE;
   STATUS[740].EXT.AlarmFailUnAck := FALSE;
   STATUS[740].Status := 0;
   STATUS[740].TimeStamp := 16#0000;
   STATUS[741].VALUE := 0.0;
   STATUS[741].TRIGVALUE := 0.0;
   STATUS[741].EXT.AlarmWarnUnAck := FALSE;
   STATUS[741].EXT.AckRequired := FALSE;
   STATUS[741].EXT.Maintanence := FALSE;
   STATUS[741].EXT.Operation := FALSE;
   STATUS[741].EXT.Forced := FALSE;
   STATUS[741].EXT.BIT29 := FALSE;
   STATUS[741].EXT.BIT30 := FALSE;
   STATUS[741].EXT.BIT31 := FALSE;
   STATUS[741].EXT.ModeBit1 := FALSE;
   STATUS[741].EXT.ModeBit2 := FALSE;
   STATUS[741].EXT.ModeBit3 := FALSE;
   STATUS[741].EXT.BIT19 := FALSE;
   STATUS[741].EXT.BIT20 := FALSE;
   STATUS[741].EXT.AlarmSuppressed := FALSE;
   STATUS[741].EXT.AlarmPrsent := FALSE;
   STATUS[741].EXT.AlarmFailUnAck := FALSE;
   STATUS[741].Status := 0;
   STATUS[741].TimeStamp := 16#0000;
   STATUS[742].VALUE := 0.0;
   STATUS[742].TRIGVALUE := 0.0;
   STATUS[742].EXT.AlarmWarnUnAck := FALSE;
   STATUS[742].EXT.AckRequired := FALSE;
   STATUS[742].EXT.Maintanence := FALSE;
   STATUS[742].EXT.Operation := FALSE;
   STATUS[742].EXT.Forced := FALSE;
   STATUS[742].EXT.BIT29 := FALSE;
   STATUS[742].EXT.BIT30 := FALSE;
   STATUS[742].EXT.BIT31 := FALSE;
   STATUS[742].EXT.ModeBit1 := FALSE;
   STATUS[742].EXT.ModeBit2 := FALSE;
   STATUS[742].EXT.ModeBit3 := FALSE;
   STATUS[742].EXT.BIT19 := FALSE;
   STATUS[742].EXT.BIT20 := FALSE;
   STATUS[742].EXT.AlarmSuppressed := FALSE;
   STATUS[742].EXT.AlarmPrsent := FALSE;
   STATUS[742].EXT.AlarmFailUnAck := FALSE;
   STATUS[742].Status := 0;
   STATUS[742].TimeStamp := 16#0000;
   STATUS[743].VALUE := 0.0;
   STATUS[743].TRIGVALUE := 0.0;
   STATUS[743].EXT.AlarmWarnUnAck := FALSE;
   STATUS[743].EXT.AckRequired := FALSE;
   STATUS[743].EXT.Maintanence := FALSE;
   STATUS[743].EXT.Operation := FALSE;
   STATUS[743].EXT.Forced := FALSE;
   STATUS[743].EXT.BIT29 := FALSE;
   STATUS[743].EXT.BIT30 := FALSE;
   STATUS[743].EXT.BIT31 := FALSE;
   STATUS[743].EXT.ModeBit1 := FALSE;
   STATUS[743].EXT.ModeBit2 := FALSE;
   STATUS[743].EXT.ModeBit3 := FALSE;
   STATUS[743].EXT.BIT19 := FALSE;
   STATUS[743].EXT.BIT20 := FALSE;
   STATUS[743].EXT.AlarmSuppressed := FALSE;
   STATUS[743].EXT.AlarmPrsent := FALSE;
   STATUS[743].EXT.AlarmFailUnAck := FALSE;
   STATUS[743].Status := 0;
   STATUS[743].TimeStamp := 16#0000;
   STATUS[744].VALUE := 0.0;
   STATUS[744].TRIGVALUE := 0.0;
   STATUS[744].EXT.AlarmWarnUnAck := FALSE;
   STATUS[744].EXT.AckRequired := FALSE;
   STATUS[744].EXT.Maintanence := FALSE;
   STATUS[744].EXT.Operation := FALSE;
   STATUS[744].EXT.Forced := FALSE;
   STATUS[744].EXT.BIT29 := FALSE;
   STATUS[744].EXT.BIT30 := FALSE;
   STATUS[744].EXT.BIT31 := FALSE;
   STATUS[744].EXT.ModeBit1 := FALSE;
   STATUS[744].EXT.ModeBit2 := FALSE;
   STATUS[744].EXT.ModeBit3 := FALSE;
   STATUS[744].EXT.BIT19 := FALSE;
   STATUS[744].EXT.BIT20 := FALSE;
   STATUS[744].EXT.AlarmSuppressed := FALSE;
   STATUS[744].EXT.AlarmPrsent := FALSE;
   STATUS[744].EXT.AlarmFailUnAck := FALSE;
   STATUS[744].Status := 0;
   STATUS[744].TimeStamp := 16#0000;
   STATUS[745].VALUE := 0.0;
   STATUS[745].TRIGVALUE := 0.0;
   STATUS[745].EXT.AlarmWarnUnAck := FALSE;
   STATUS[745].EXT.AckRequired := FALSE;
   STATUS[745].EXT.Maintanence := FALSE;
   STATUS[745].EXT.Operation := FALSE;
   STATUS[745].EXT.Forced := FALSE;
   STATUS[745].EXT.BIT29 := FALSE;
   STATUS[745].EXT.BIT30 := FALSE;
   STATUS[745].EXT.BIT31 := FALSE;
   STATUS[745].EXT.ModeBit1 := FALSE;
   STATUS[745].EXT.ModeBit2 := FALSE;
   STATUS[745].EXT.ModeBit3 := FALSE;
   STATUS[745].EXT.BIT19 := FALSE;
   STATUS[745].EXT.BIT20 := FALSE;
   STATUS[745].EXT.AlarmSuppressed := FALSE;
   STATUS[745].EXT.AlarmPrsent := FALSE;
   STATUS[745].EXT.AlarmFailUnAck := FALSE;
   STATUS[745].Status := 0;
   STATUS[745].TimeStamp := 16#0000;
   STATUS[746].VALUE := 0.0;
   STATUS[746].TRIGVALUE := 0.0;
   STATUS[746].EXT.AlarmWarnUnAck := FALSE;
   STATUS[746].EXT.AckRequired := FALSE;
   STATUS[746].EXT.Maintanence := FALSE;
   STATUS[746].EXT.Operation := FALSE;
   STATUS[746].EXT.Forced := FALSE;
   STATUS[746].EXT.BIT29 := FALSE;
   STATUS[746].EXT.BIT30 := FALSE;
   STATUS[746].EXT.BIT31 := FALSE;
   STATUS[746].EXT.ModeBit1 := FALSE;
   STATUS[746].EXT.ModeBit2 := FALSE;
   STATUS[746].EXT.ModeBit3 := FALSE;
   STATUS[746].EXT.BIT19 := FALSE;
   STATUS[746].EXT.BIT20 := FALSE;
   STATUS[746].EXT.AlarmSuppressed := FALSE;
   STATUS[746].EXT.AlarmPrsent := FALSE;
   STATUS[746].EXT.AlarmFailUnAck := FALSE;
   STATUS[746].Status := 0;
   STATUS[746].TimeStamp := 16#0000;
   STATUS[747].VALUE := 0.0;
   STATUS[747].TRIGVALUE := 0.0;
   STATUS[747].EXT.AlarmWarnUnAck := FALSE;
   STATUS[747].EXT.AckRequired := FALSE;
   STATUS[747].EXT.Maintanence := FALSE;
   STATUS[747].EXT.Operation := FALSE;
   STATUS[747].EXT.Forced := FALSE;
   STATUS[747].EXT.BIT29 := FALSE;
   STATUS[747].EXT.BIT30 := FALSE;
   STATUS[747].EXT.BIT31 := FALSE;
   STATUS[747].EXT.ModeBit1 := FALSE;
   STATUS[747].EXT.ModeBit2 := FALSE;
   STATUS[747].EXT.ModeBit3 := FALSE;
   STATUS[747].EXT.BIT19 := FALSE;
   STATUS[747].EXT.BIT20 := FALSE;
   STATUS[747].EXT.AlarmSuppressed := FALSE;
   STATUS[747].EXT.AlarmPrsent := FALSE;
   STATUS[747].EXT.AlarmFailUnAck := FALSE;
   STATUS[747].Status := 0;
   STATUS[747].TimeStamp := 16#0000;
   STATUS[748].VALUE := 0.0;
   STATUS[748].TRIGVALUE := 0.0;
   STATUS[748].EXT.AlarmWarnUnAck := FALSE;
   STATUS[748].EXT.AckRequired := FALSE;
   STATUS[748].EXT.Maintanence := FALSE;
   STATUS[748].EXT.Operation := FALSE;
   STATUS[748].EXT.Forced := FALSE;
   STATUS[748].EXT.BIT29 := FALSE;
   STATUS[748].EXT.BIT30 := FALSE;
   STATUS[748].EXT.BIT31 := FALSE;
   STATUS[748].EXT.ModeBit1 := FALSE;
   STATUS[748].EXT.ModeBit2 := FALSE;
   STATUS[748].EXT.ModeBit3 := FALSE;
   STATUS[748].EXT.BIT19 := FALSE;
   STATUS[748].EXT.BIT20 := FALSE;
   STATUS[748].EXT.AlarmSuppressed := FALSE;
   STATUS[748].EXT.AlarmPrsent := FALSE;
   STATUS[748].EXT.AlarmFailUnAck := FALSE;
   STATUS[748].Status := 0;
   STATUS[748].TimeStamp := 16#0000;
   STATUS[749].VALUE := 0.0;
   STATUS[749].TRIGVALUE := 0.0;
   STATUS[749].EXT.AlarmWarnUnAck := FALSE;
   STATUS[749].EXT.AckRequired := FALSE;
   STATUS[749].EXT.Maintanence := FALSE;
   STATUS[749].EXT.Operation := FALSE;
   STATUS[749].EXT.Forced := FALSE;
   STATUS[749].EXT.BIT29 := FALSE;
   STATUS[749].EXT.BIT30 := FALSE;
   STATUS[749].EXT.BIT31 := FALSE;
   STATUS[749].EXT.ModeBit1 := FALSE;
   STATUS[749].EXT.ModeBit2 := FALSE;
   STATUS[749].EXT.ModeBit3 := FALSE;
   STATUS[749].EXT.BIT19 := FALSE;
   STATUS[749].EXT.BIT20 := FALSE;
   STATUS[749].EXT.AlarmSuppressed := FALSE;
   STATUS[749].EXT.AlarmPrsent := FALSE;
   STATUS[749].EXT.AlarmFailUnAck := FALSE;
   STATUS[749].Status := 0;
   STATUS[749].TimeStamp := 16#0000;
   STATUS[750].VALUE := 0.0;
   STATUS[750].TRIGVALUE := 0.0;
   STATUS[750].EXT.AlarmWarnUnAck := FALSE;
   STATUS[750].EXT.AckRequired := FALSE;
   STATUS[750].EXT.Maintanence := FALSE;
   STATUS[750].EXT.Operation := FALSE;
   STATUS[750].EXT.Forced := FALSE;
   STATUS[750].EXT.BIT29 := FALSE;
   STATUS[750].EXT.BIT30 := FALSE;
   STATUS[750].EXT.BIT31 := FALSE;
   STATUS[750].EXT.ModeBit1 := FALSE;
   STATUS[750].EXT.ModeBit2 := FALSE;
   STATUS[750].EXT.ModeBit3 := FALSE;
   STATUS[750].EXT.BIT19 := FALSE;
   STATUS[750].EXT.BIT20 := FALSE;
   STATUS[750].EXT.AlarmSuppressed := FALSE;
   STATUS[750].EXT.AlarmPrsent := FALSE;
   STATUS[750].EXT.AlarmFailUnAck := FALSE;
   STATUS[750].Status := 0;
   STATUS[750].TimeStamp := 16#0000;
   STATUS[751].VALUE := 0.0;
   STATUS[751].TRIGVALUE := 0.0;
   STATUS[751].EXT.AlarmWarnUnAck := FALSE;
   STATUS[751].EXT.AckRequired := FALSE;
   STATUS[751].EXT.Maintanence := FALSE;
   STATUS[751].EXT.Operation := FALSE;
   STATUS[751].EXT.Forced := FALSE;
   STATUS[751].EXT.BIT29 := FALSE;
   STATUS[751].EXT.BIT30 := FALSE;
   STATUS[751].EXT.BIT31 := FALSE;
   STATUS[751].EXT.ModeBit1 := FALSE;
   STATUS[751].EXT.ModeBit2 := FALSE;
   STATUS[751].EXT.ModeBit3 := FALSE;
   STATUS[751].EXT.BIT19 := FALSE;
   STATUS[751].EXT.BIT20 := FALSE;
   STATUS[751].EXT.AlarmSuppressed := FALSE;
   STATUS[751].EXT.AlarmPrsent := FALSE;
   STATUS[751].EXT.AlarmFailUnAck := FALSE;
   STATUS[751].Status := 0;
   STATUS[751].TimeStamp := 16#0000;
   STATUS[752].VALUE := 0.0;
   STATUS[752].TRIGVALUE := 0.0;
   STATUS[752].EXT.AlarmWarnUnAck := FALSE;
   STATUS[752].EXT.AckRequired := FALSE;
   STATUS[752].EXT.Maintanence := FALSE;
   STATUS[752].EXT.Operation := FALSE;
   STATUS[752].EXT.Forced := FALSE;
   STATUS[752].EXT.BIT29 := FALSE;
   STATUS[752].EXT.BIT30 := FALSE;
   STATUS[752].EXT.BIT31 := FALSE;
   STATUS[752].EXT.ModeBit1 := FALSE;
   STATUS[752].EXT.ModeBit2 := FALSE;
   STATUS[752].EXT.ModeBit3 := FALSE;
   STATUS[752].EXT.BIT19 := FALSE;
   STATUS[752].EXT.BIT20 := FALSE;
   STATUS[752].EXT.AlarmSuppressed := FALSE;
   STATUS[752].EXT.AlarmPrsent := FALSE;
   STATUS[752].EXT.AlarmFailUnAck := FALSE;
   STATUS[752].Status := 0;
   STATUS[752].TimeStamp := 16#0000;
   STATUS[753].VALUE := 0.0;
   STATUS[753].TRIGVALUE := 0.0;
   STATUS[753].EXT.AlarmWarnUnAck := FALSE;
   STATUS[753].EXT.AckRequired := FALSE;
   STATUS[753].EXT.Maintanence := FALSE;
   STATUS[753].EXT.Operation := FALSE;
   STATUS[753].EXT.Forced := FALSE;
   STATUS[753].EXT.BIT29 := FALSE;
   STATUS[753].EXT.BIT30 := FALSE;
   STATUS[753].EXT.BIT31 := FALSE;
   STATUS[753].EXT.ModeBit1 := FALSE;
   STATUS[753].EXT.ModeBit2 := FALSE;
   STATUS[753].EXT.ModeBit3 := FALSE;
   STATUS[753].EXT.BIT19 := FALSE;
   STATUS[753].EXT.BIT20 := FALSE;
   STATUS[753].EXT.AlarmSuppressed := FALSE;
   STATUS[753].EXT.AlarmPrsent := FALSE;
   STATUS[753].EXT.AlarmFailUnAck := FALSE;
   STATUS[753].Status := 0;
   STATUS[753].TimeStamp := 16#0000;
   STATUS[754].VALUE := 0.0;
   STATUS[754].TRIGVALUE := 0.0;
   STATUS[754].EXT.AlarmWarnUnAck := FALSE;
   STATUS[754].EXT.AckRequired := FALSE;
   STATUS[754].EXT.Maintanence := FALSE;
   STATUS[754].EXT.Operation := FALSE;
   STATUS[754].EXT.Forced := FALSE;
   STATUS[754].EXT.BIT29 := FALSE;
   STATUS[754].EXT.BIT30 := FALSE;
   STATUS[754].EXT.BIT31 := FALSE;
   STATUS[754].EXT.ModeBit1 := FALSE;
   STATUS[754].EXT.ModeBit2 := FALSE;
   STATUS[754].EXT.ModeBit3 := FALSE;
   STATUS[754].EXT.BIT19 := FALSE;
   STATUS[754].EXT.BIT20 := FALSE;
   STATUS[754].EXT.AlarmSuppressed := FALSE;
   STATUS[754].EXT.AlarmPrsent := FALSE;
   STATUS[754].EXT.AlarmFailUnAck := FALSE;
   STATUS[754].Status := 0;
   STATUS[754].TimeStamp := 16#0000;
   STATUS[755].VALUE := 0.0;
   STATUS[755].TRIGVALUE := 0.0;
   STATUS[755].EXT.AlarmWarnUnAck := FALSE;
   STATUS[755].EXT.AckRequired := FALSE;
   STATUS[755].EXT.Maintanence := FALSE;
   STATUS[755].EXT.Operation := FALSE;
   STATUS[755].EXT.Forced := FALSE;
   STATUS[755].EXT.BIT29 := FALSE;
   STATUS[755].EXT.BIT30 := FALSE;
   STATUS[755].EXT.BIT31 := FALSE;
   STATUS[755].EXT.ModeBit1 := FALSE;
   STATUS[755].EXT.ModeBit2 := FALSE;
   STATUS[755].EXT.ModeBit3 := FALSE;
   STATUS[755].EXT.BIT19 := FALSE;
   STATUS[755].EXT.BIT20 := FALSE;
   STATUS[755].EXT.AlarmSuppressed := FALSE;
   STATUS[755].EXT.AlarmPrsent := FALSE;
   STATUS[755].EXT.AlarmFailUnAck := FALSE;
   STATUS[755].Status := 0;
   STATUS[755].TimeStamp := 16#0000;
   STATUS[756].VALUE := 0.0;
   STATUS[756].TRIGVALUE := 0.0;
   STATUS[756].EXT.AlarmWarnUnAck := FALSE;
   STATUS[756].EXT.AckRequired := FALSE;
   STATUS[756].EXT.Maintanence := FALSE;
   STATUS[756].EXT.Operation := FALSE;
   STATUS[756].EXT.Forced := FALSE;
   STATUS[756].EXT.BIT29 := FALSE;
   STATUS[756].EXT.BIT30 := FALSE;
   STATUS[756].EXT.BIT31 := FALSE;
   STATUS[756].EXT.ModeBit1 := FALSE;
   STATUS[756].EXT.ModeBit2 := FALSE;
   STATUS[756].EXT.ModeBit3 := FALSE;
   STATUS[756].EXT.BIT19 := FALSE;
   STATUS[756].EXT.BIT20 := FALSE;
   STATUS[756].EXT.AlarmSuppressed := FALSE;
   STATUS[756].EXT.AlarmPrsent := FALSE;
   STATUS[756].EXT.AlarmFailUnAck := FALSE;
   STATUS[756].Status := 0;
   STATUS[756].TimeStamp := 16#0000;
   STATUS[757].VALUE := 0.0;
   STATUS[757].TRIGVALUE := 0.0;
   STATUS[757].EXT.AlarmWarnUnAck := FALSE;
   STATUS[757].EXT.AckRequired := FALSE;
   STATUS[757].EXT.Maintanence := FALSE;
   STATUS[757].EXT.Operation := FALSE;
   STATUS[757].EXT.Forced := FALSE;
   STATUS[757].EXT.BIT29 := FALSE;
   STATUS[757].EXT.BIT30 := FALSE;
   STATUS[757].EXT.BIT31 := FALSE;
   STATUS[757].EXT.ModeBit1 := FALSE;
   STATUS[757].EXT.ModeBit2 := FALSE;
   STATUS[757].EXT.ModeBit3 := FALSE;
   STATUS[757].EXT.BIT19 := FALSE;
   STATUS[757].EXT.BIT20 := FALSE;
   STATUS[757].EXT.AlarmSuppressed := FALSE;
   STATUS[757].EXT.AlarmPrsent := FALSE;
   STATUS[757].EXT.AlarmFailUnAck := FALSE;
   STATUS[757].Status := 0;
   STATUS[757].TimeStamp := 16#0000;
   STATUS[758].VALUE := 0.0;
   STATUS[758].TRIGVALUE := 0.0;
   STATUS[758].EXT.AlarmWarnUnAck := FALSE;
   STATUS[758].EXT.AckRequired := FALSE;
   STATUS[758].EXT.Maintanence := FALSE;
   STATUS[758].EXT.Operation := FALSE;
   STATUS[758].EXT.Forced := FALSE;
   STATUS[758].EXT.BIT29 := FALSE;
   STATUS[758].EXT.BIT30 := FALSE;
   STATUS[758].EXT.BIT31 := FALSE;
   STATUS[758].EXT.ModeBit1 := FALSE;
   STATUS[758].EXT.ModeBit2 := FALSE;
   STATUS[758].EXT.ModeBit3 := FALSE;
   STATUS[758].EXT.BIT19 := FALSE;
   STATUS[758].EXT.BIT20 := FALSE;
   STATUS[758].EXT.AlarmSuppressed := FALSE;
   STATUS[758].EXT.AlarmPrsent := FALSE;
   STATUS[758].EXT.AlarmFailUnAck := FALSE;
   STATUS[758].Status := 0;
   STATUS[758].TimeStamp := 16#0000;
   STATUS[759].VALUE := 0.0;
   STATUS[759].TRIGVALUE := 0.0;
   STATUS[759].EXT.AlarmWarnUnAck := FALSE;
   STATUS[759].EXT.AckRequired := FALSE;
   STATUS[759].EXT.Maintanence := FALSE;
   STATUS[759].EXT.Operation := FALSE;
   STATUS[759].EXT.Forced := FALSE;
   STATUS[759].EXT.BIT29 := FALSE;
   STATUS[759].EXT.BIT30 := FALSE;
   STATUS[759].EXT.BIT31 := FALSE;
   STATUS[759].EXT.ModeBit1 := FALSE;
   STATUS[759].EXT.ModeBit2 := FALSE;
   STATUS[759].EXT.ModeBit3 := FALSE;
   STATUS[759].EXT.BIT19 := FALSE;
   STATUS[759].EXT.BIT20 := FALSE;
   STATUS[759].EXT.AlarmSuppressed := FALSE;
   STATUS[759].EXT.AlarmPrsent := FALSE;
   STATUS[759].EXT.AlarmFailUnAck := FALSE;
   STATUS[759].Status := 0;
   STATUS[759].TimeStamp := 16#0000;
   STATUS[760].VALUE := 0.0;
   STATUS[760].TRIGVALUE := 0.0;
   STATUS[760].EXT.AlarmWarnUnAck := FALSE;
   STATUS[760].EXT.AckRequired := FALSE;
   STATUS[760].EXT.Maintanence := FALSE;
   STATUS[760].EXT.Operation := FALSE;
   STATUS[760].EXT.Forced := FALSE;
   STATUS[760].EXT.BIT29 := FALSE;
   STATUS[760].EXT.BIT30 := FALSE;
   STATUS[760].EXT.BIT31 := FALSE;
   STATUS[760].EXT.ModeBit1 := FALSE;
   STATUS[760].EXT.ModeBit2 := FALSE;
   STATUS[760].EXT.ModeBit3 := FALSE;
   STATUS[760].EXT.BIT19 := FALSE;
   STATUS[760].EXT.BIT20 := FALSE;
   STATUS[760].EXT.AlarmSuppressed := FALSE;
   STATUS[760].EXT.AlarmPrsent := FALSE;
   STATUS[760].EXT.AlarmFailUnAck := FALSE;
   STATUS[760].Status := 0;
   STATUS[760].TimeStamp := 16#0000;
   STATUS[761].VALUE := 0.0;
   STATUS[761].TRIGVALUE := 0.0;
   STATUS[761].EXT.AlarmWarnUnAck := FALSE;
   STATUS[761].EXT.AckRequired := FALSE;
   STATUS[761].EXT.Maintanence := FALSE;
   STATUS[761].EXT.Operation := FALSE;
   STATUS[761].EXT.Forced := FALSE;
   STATUS[761].EXT.BIT29 := FALSE;
   STATUS[761].EXT.BIT30 := FALSE;
   STATUS[761].EXT.BIT31 := FALSE;
   STATUS[761].EXT.ModeBit1 := FALSE;
   STATUS[761].EXT.ModeBit2 := FALSE;
   STATUS[761].EXT.ModeBit3 := FALSE;
   STATUS[761].EXT.BIT19 := FALSE;
   STATUS[761].EXT.BIT20 := FALSE;
   STATUS[761].EXT.AlarmSuppressed := FALSE;
   STATUS[761].EXT.AlarmPrsent := FALSE;
   STATUS[761].EXT.AlarmFailUnAck := FALSE;
   STATUS[761].Status := 0;
   STATUS[761].TimeStamp := 16#0000;
   STATUS[762].VALUE := 0.0;
   STATUS[762].TRIGVALUE := 0.0;
   STATUS[762].EXT.AlarmWarnUnAck := FALSE;
   STATUS[762].EXT.AckRequired := FALSE;
   STATUS[762].EXT.Maintanence := FALSE;
   STATUS[762].EXT.Operation := FALSE;
   STATUS[762].EXT.Forced := FALSE;
   STATUS[762].EXT.BIT29 := FALSE;
   STATUS[762].EXT.BIT30 := FALSE;
   STATUS[762].EXT.BIT31 := FALSE;
   STATUS[762].EXT.ModeBit1 := FALSE;
   STATUS[762].EXT.ModeBit2 := FALSE;
   STATUS[762].EXT.ModeBit3 := FALSE;
   STATUS[762].EXT.BIT19 := FALSE;
   STATUS[762].EXT.BIT20 := FALSE;
   STATUS[762].EXT.AlarmSuppressed := FALSE;
   STATUS[762].EXT.AlarmPrsent := FALSE;
   STATUS[762].EXT.AlarmFailUnAck := FALSE;
   STATUS[762].Status := 0;
   STATUS[762].TimeStamp := 16#0000;
   STATUS[763].VALUE := 0.0;
   STATUS[763].TRIGVALUE := 0.0;
   STATUS[763].EXT.AlarmWarnUnAck := FALSE;
   STATUS[763].EXT.AckRequired := FALSE;
   STATUS[763].EXT.Maintanence := FALSE;
   STATUS[763].EXT.Operation := FALSE;
   STATUS[763].EXT.Forced := FALSE;
   STATUS[763].EXT.BIT29 := FALSE;
   STATUS[763].EXT.BIT30 := FALSE;
   STATUS[763].EXT.BIT31 := FALSE;
   STATUS[763].EXT.ModeBit1 := FALSE;
   STATUS[763].EXT.ModeBit2 := FALSE;
   STATUS[763].EXT.ModeBit3 := FALSE;
   STATUS[763].EXT.BIT19 := FALSE;
   STATUS[763].EXT.BIT20 := FALSE;
   STATUS[763].EXT.AlarmSuppressed := FALSE;
   STATUS[763].EXT.AlarmPrsent := FALSE;
   STATUS[763].EXT.AlarmFailUnAck := FALSE;
   STATUS[763].Status := 0;
   STATUS[763].TimeStamp := 16#0000;
   STATUS[764].VALUE := 0.0;
   STATUS[764].TRIGVALUE := 0.0;
   STATUS[764].EXT.AlarmWarnUnAck := FALSE;
   STATUS[764].EXT.AckRequired := FALSE;
   STATUS[764].EXT.Maintanence := FALSE;
   STATUS[764].EXT.Operation := FALSE;
   STATUS[764].EXT.Forced := FALSE;
   STATUS[764].EXT.BIT29 := FALSE;
   STATUS[764].EXT.BIT30 := FALSE;
   STATUS[764].EXT.BIT31 := FALSE;
   STATUS[764].EXT.ModeBit1 := FALSE;
   STATUS[764].EXT.ModeBit2 := FALSE;
   STATUS[764].EXT.ModeBit3 := FALSE;
   STATUS[764].EXT.BIT19 := FALSE;
   STATUS[764].EXT.BIT20 := FALSE;
   STATUS[764].EXT.AlarmSuppressed := FALSE;
   STATUS[764].EXT.AlarmPrsent := FALSE;
   STATUS[764].EXT.AlarmFailUnAck := FALSE;
   STATUS[764].Status := 0;
   STATUS[764].TimeStamp := 16#0000;
   STATUS[765].VALUE := 0.0;
   STATUS[765].TRIGVALUE := 0.0;
   STATUS[765].EXT.AlarmWarnUnAck := FALSE;
   STATUS[765].EXT.AckRequired := FALSE;
   STATUS[765].EXT.Maintanence := FALSE;
   STATUS[765].EXT.Operation := FALSE;
   STATUS[765].EXT.Forced := FALSE;
   STATUS[765].EXT.BIT29 := FALSE;
   STATUS[765].EXT.BIT30 := FALSE;
   STATUS[765].EXT.BIT31 := FALSE;
   STATUS[765].EXT.ModeBit1 := FALSE;
   STATUS[765].EXT.ModeBit2 := FALSE;
   STATUS[765].EXT.ModeBit3 := FALSE;
   STATUS[765].EXT.BIT19 := FALSE;
   STATUS[765].EXT.BIT20 := FALSE;
   STATUS[765].EXT.AlarmSuppressed := FALSE;
   STATUS[765].EXT.AlarmPrsent := FALSE;
   STATUS[765].EXT.AlarmFailUnAck := FALSE;
   STATUS[765].Status := 0;
   STATUS[765].TimeStamp := 16#0000;
   STATUS[766].VALUE := 0.0;
   STATUS[766].TRIGVALUE := 0.0;
   STATUS[766].EXT.AlarmWarnUnAck := FALSE;
   STATUS[766].EXT.AckRequired := FALSE;
   STATUS[766].EXT.Maintanence := FALSE;
   STATUS[766].EXT.Operation := FALSE;
   STATUS[766].EXT.Forced := FALSE;
   STATUS[766].EXT.BIT29 := FALSE;
   STATUS[766].EXT.BIT30 := FALSE;
   STATUS[766].EXT.BIT31 := FALSE;
   STATUS[766].EXT.ModeBit1 := FALSE;
   STATUS[766].EXT.ModeBit2 := FALSE;
   STATUS[766].EXT.ModeBit3 := FALSE;
   STATUS[766].EXT.BIT19 := FALSE;
   STATUS[766].EXT.BIT20 := FALSE;
   STATUS[766].EXT.AlarmSuppressed := FALSE;
   STATUS[766].EXT.AlarmPrsent := FALSE;
   STATUS[766].EXT.AlarmFailUnAck := FALSE;
   STATUS[766].Status := 0;
   STATUS[766].TimeStamp := 16#0000;
   STATUS[767].VALUE := 0.0;
   STATUS[767].TRIGVALUE := 0.0;
   STATUS[767].EXT.AlarmWarnUnAck := FALSE;
   STATUS[767].EXT.AckRequired := FALSE;
   STATUS[767].EXT.Maintanence := FALSE;
   STATUS[767].EXT.Operation := FALSE;
   STATUS[767].EXT.Forced := FALSE;
   STATUS[767].EXT.BIT29 := FALSE;
   STATUS[767].EXT.BIT30 := FALSE;
   STATUS[767].EXT.BIT31 := FALSE;
   STATUS[767].EXT.ModeBit1 := FALSE;
   STATUS[767].EXT.ModeBit2 := FALSE;
   STATUS[767].EXT.ModeBit3 := FALSE;
   STATUS[767].EXT.BIT19 := FALSE;
   STATUS[767].EXT.BIT20 := FALSE;
   STATUS[767].EXT.AlarmSuppressed := FALSE;
   STATUS[767].EXT.AlarmPrsent := FALSE;
   STATUS[767].EXT.AlarmFailUnAck := FALSE;
   STATUS[767].Status := 0;
   STATUS[767].TimeStamp := 16#0000;
   STATUS[768].VALUE := 0.0;
   STATUS[768].TRIGVALUE := 0.0;
   STATUS[768].EXT.AlarmWarnUnAck := FALSE;
   STATUS[768].EXT.AckRequired := FALSE;
   STATUS[768].EXT.Maintanence := FALSE;
   STATUS[768].EXT.Operation := FALSE;
   STATUS[768].EXT.Forced := FALSE;
   STATUS[768].EXT.BIT29 := FALSE;
   STATUS[768].EXT.BIT30 := FALSE;
   STATUS[768].EXT.BIT31 := FALSE;
   STATUS[768].EXT.ModeBit1 := FALSE;
   STATUS[768].EXT.ModeBit2 := FALSE;
   STATUS[768].EXT.ModeBit3 := FALSE;
   STATUS[768].EXT.BIT19 := FALSE;
   STATUS[768].EXT.BIT20 := FALSE;
   STATUS[768].EXT.AlarmSuppressed := FALSE;
   STATUS[768].EXT.AlarmPrsent := FALSE;
   STATUS[768].EXT.AlarmFailUnAck := FALSE;
   STATUS[768].Status := 0;
   STATUS[768].TimeStamp := 16#0000;
   STATUS[769].VALUE := 0.0;
   STATUS[769].TRIGVALUE := 0.0;
   STATUS[769].EXT.AlarmWarnUnAck := FALSE;
   STATUS[769].EXT.AckRequired := FALSE;
   STATUS[769].EXT.Maintanence := FALSE;
   STATUS[769].EXT.Operation := FALSE;
   STATUS[769].EXT.Forced := FALSE;
   STATUS[769].EXT.BIT29 := FALSE;
   STATUS[769].EXT.BIT30 := FALSE;
   STATUS[769].EXT.BIT31 := FALSE;
   STATUS[769].EXT.ModeBit1 := FALSE;
   STATUS[769].EXT.ModeBit2 := FALSE;
   STATUS[769].EXT.ModeBit3 := FALSE;
   STATUS[769].EXT.BIT19 := FALSE;
   STATUS[769].EXT.BIT20 := FALSE;
   STATUS[769].EXT.AlarmSuppressed := FALSE;
   STATUS[769].EXT.AlarmPrsent := FALSE;
   STATUS[769].EXT.AlarmFailUnAck := FALSE;
   STATUS[769].Status := 0;
   STATUS[769].TimeStamp := 16#0000;
   STATUS[770].VALUE := 0.0;
   STATUS[770].TRIGVALUE := 0.0;
   STATUS[770].EXT.AlarmWarnUnAck := FALSE;
   STATUS[770].EXT.AckRequired := FALSE;
   STATUS[770].EXT.Maintanence := FALSE;
   STATUS[770].EXT.Operation := FALSE;
   STATUS[770].EXT.Forced := FALSE;
   STATUS[770].EXT.BIT29 := FALSE;
   STATUS[770].EXT.BIT30 := FALSE;
   STATUS[770].EXT.BIT31 := FALSE;
   STATUS[770].EXT.ModeBit1 := FALSE;
   STATUS[770].EXT.ModeBit2 := FALSE;
   STATUS[770].EXT.ModeBit3 := FALSE;
   STATUS[770].EXT.BIT19 := FALSE;
   STATUS[770].EXT.BIT20 := FALSE;
   STATUS[770].EXT.AlarmSuppressed := FALSE;
   STATUS[770].EXT.AlarmPrsent := FALSE;
   STATUS[770].EXT.AlarmFailUnAck := FALSE;
   STATUS[770].Status := 0;
   STATUS[770].TimeStamp := 16#0000;
   STATUS[771].VALUE := 0.0;
   STATUS[771].TRIGVALUE := 0.0;
   STATUS[771].EXT.AlarmWarnUnAck := FALSE;
   STATUS[771].EXT.AckRequired := FALSE;
   STATUS[771].EXT.Maintanence := FALSE;
   STATUS[771].EXT.Operation := FALSE;
   STATUS[771].EXT.Forced := FALSE;
   STATUS[771].EXT.BIT29 := FALSE;
   STATUS[771].EXT.BIT30 := FALSE;
   STATUS[771].EXT.BIT31 := FALSE;
   STATUS[771].EXT.ModeBit1 := FALSE;
   STATUS[771].EXT.ModeBit2 := FALSE;
   STATUS[771].EXT.ModeBit3 := FALSE;
   STATUS[771].EXT.BIT19 := FALSE;
   STATUS[771].EXT.BIT20 := FALSE;
   STATUS[771].EXT.AlarmSuppressed := FALSE;
   STATUS[771].EXT.AlarmPrsent := FALSE;
   STATUS[771].EXT.AlarmFailUnAck := FALSE;
   STATUS[771].Status := 0;
   STATUS[771].TimeStamp := 16#0000;
   STATUS[772].VALUE := 0.0;
   STATUS[772].TRIGVALUE := 0.0;
   STATUS[772].EXT.AlarmWarnUnAck := FALSE;
   STATUS[772].EXT.AckRequired := FALSE;
   STATUS[772].EXT.Maintanence := FALSE;
   STATUS[772].EXT.Operation := FALSE;
   STATUS[772].EXT.Forced := FALSE;
   STATUS[772].EXT.BIT29 := FALSE;
   STATUS[772].EXT.BIT30 := FALSE;
   STATUS[772].EXT.BIT31 := FALSE;
   STATUS[772].EXT.ModeBit1 := FALSE;
   STATUS[772].EXT.ModeBit2 := FALSE;
   STATUS[772].EXT.ModeBit3 := FALSE;
   STATUS[772].EXT.BIT19 := FALSE;
   STATUS[772].EXT.BIT20 := FALSE;
   STATUS[772].EXT.AlarmSuppressed := FALSE;
   STATUS[772].EXT.AlarmPrsent := FALSE;
   STATUS[772].EXT.AlarmFailUnAck := FALSE;
   STATUS[772].Status := 0;
   STATUS[772].TimeStamp := 16#0000;
   STATUS[773].VALUE := 0.0;
   STATUS[773].TRIGVALUE := 0.0;
   STATUS[773].EXT.AlarmWarnUnAck := FALSE;
   STATUS[773].EXT.AckRequired := FALSE;
   STATUS[773].EXT.Maintanence := FALSE;
   STATUS[773].EXT.Operation := FALSE;
   STATUS[773].EXT.Forced := FALSE;
   STATUS[773].EXT.BIT29 := FALSE;
   STATUS[773].EXT.BIT30 := FALSE;
   STATUS[773].EXT.BIT31 := FALSE;
   STATUS[773].EXT.ModeBit1 := FALSE;
   STATUS[773].EXT.ModeBit2 := FALSE;
   STATUS[773].EXT.ModeBit3 := FALSE;
   STATUS[773].EXT.BIT19 := FALSE;
   STATUS[773].EXT.BIT20 := FALSE;
   STATUS[773].EXT.AlarmSuppressed := FALSE;
   STATUS[773].EXT.AlarmPrsent := FALSE;
   STATUS[773].EXT.AlarmFailUnAck := FALSE;
   STATUS[773].Status := 0;
   STATUS[773].TimeStamp := 16#0000;
   STATUS[774].VALUE := 0.0;
   STATUS[774].TRIGVALUE := 0.0;
   STATUS[774].EXT.AlarmWarnUnAck := FALSE;
   STATUS[774].EXT.AckRequired := FALSE;
   STATUS[774].EXT.Maintanence := FALSE;
   STATUS[774].EXT.Operation := FALSE;
   STATUS[774].EXT.Forced := FALSE;
   STATUS[774].EXT.BIT29 := FALSE;
   STATUS[774].EXT.BIT30 := FALSE;
   STATUS[774].EXT.BIT31 := FALSE;
   STATUS[774].EXT.ModeBit1 := FALSE;
   STATUS[774].EXT.ModeBit2 := FALSE;
   STATUS[774].EXT.ModeBit3 := FALSE;
